KUKA KRL program: EPS_2_25990_SANMH02_A_20251014015154.src

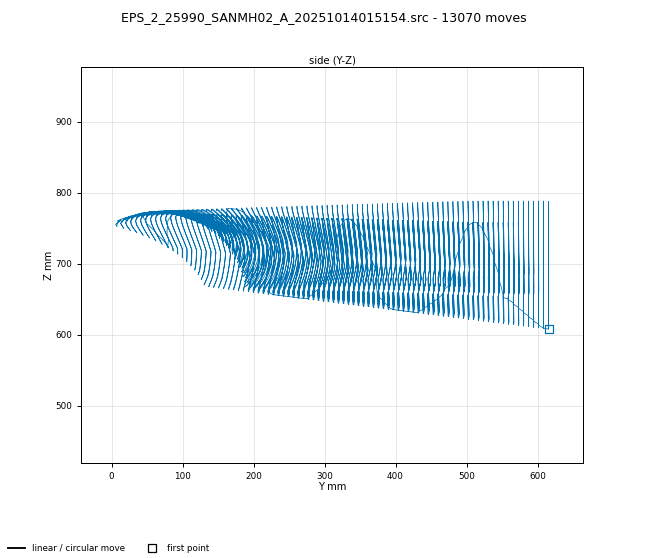
[picture p0: tool path of EPS_2_25990_SANMH02_A_20251014015154.src, 13070 of 13072 moves have a stored position in this frame; points joined in program order, loops and branches not executed]
&ACCESS RVP
&REL 4
&COMMENT QRS 19112012
&PARAM EDITMASK = *
DEF PART()
EXT BAS (BAS_COMMAND :IN,REAL :IN )
INT I
BAS (#INITMOV,0 )

;KUKA QRS Post kuka4.cps  Date:22-06-2017 !

File_ID=2883

QRS_PRE_INIT()

;Init var - Until changes are made in qrs_pre_init
Outlet_Square_prg=0
Inlet_1_Square_prg=0
Inlet_2_Square_prg=0
Inlet_3_Square_prg=0
Inlet_4_Square_prg=0
Inlet_5_Square_prg=0

Outlet_1={X 0.000, Y 504.220, Z 687.500, B 0.000, E1 0.000 }
Inlet_1={X 0.000, Y 506.400, Z 657.500, B 0.000, E1 135.000 }
Inlet_2={X 0.000, Y 506.400, Z 657.500, B 0.000, E1 224.000 }
Outlet_1_type=201
Inlet_1_type=201
Inlet_2_type=201
;QRS#1=Sidecore dimensions
;QRS#2=200-8" PVC SDR 35
;QRS#3=200-8" PVC SDR 35
;QRS#4=200-8" PVC SDR 35
;QRS#5=
;QRS#6=
;QRS#7=
;QRS#8=
;QRS#9=12-08 PSX
;QRS#10=12-08 PSX
;QRS#11=12-08 PSX
;QRS#12=
;QRS#13=
;QRS#14=
;QRS#15=
;QRS#16=1220x127x1067 3,5'
;QRS#17=EPS Height
;QRS#18=788
;QRS#19=*
;QRS#20= UPDATED VERSION 22-06-2017
;QRS#21=*
Outlet_Square=0100
Inlet_1_Square=0100
Inlet_2_Square=0100
Inlet_3_Square=0
Inlet_4_Square=0
Inlet_5_Square=0
Mill_Square=1
Outlet_Square_Prg=204
Inlet_1_Square_prg=204
Inlet_2_Square_prg=204

QRS_INIT()

$ADVANCE=5

; T1
PTP {E1 173.417,E2 173.417}
PTP {X 0,Y 615.493,A -85,B 0,C 180,E1 173.417,E2 173.417,E3 0,E4 0,E5 0,E6 0}
QRS_SPEED_INIT()
LIN {X 0,Y 615.493,Z 607.697,A -85,B 0,C 180,E1 173.417,E2 173.417,E3 0,E4 0,E5 0,E6 0} C_VEL
LIN {X 0,Y 615.492,Z 607.697,A -85,B 0,C 180,E1 170.801,E2 170.801} C_VEL
LIN {X 0,Y 615.497,Z 607.973,A -85,B 0,C 180,E1 170.138,E2 170.138} C_VEL
LIN {X 0,Y 615.488,Z 612.63,A -85,B 0,C 180,E1 167.47,E2 167.47} C_VEL
LIN {X 0,Y 615.489,Z 617.473,A -85,B 0,C 180,E1 164.774,E2 164.774} C_VEL
LIN {X 0,Y 615.454,Z 622.534,A -85,B 0,C 180,E1 162.042,E2 162.042} C_VEL
LIN {X 0,Y 615.492,Z 627.771,A -85,B 0,C 180,E1 159.269,E2 159.269} C_VEL
LIN {X 0,Y 615.481,Z 633.246,A -85,B 0,C 180,E1 156.443,E2 156.443} C_VEL
LIN {X 0,Y 615.483,Z 637.503,A -85,B 0,C 180,E1 154.284,E2 154.284} C_VEL
LIN {X 0,Y 615.478,Z 642.947,A -85,B 0,C 180,E1 151.551,E2 151.551} C_VEL
LIN {X 0,Y 615.49,Z 648.292,A -85,B 0,C 180,E1 148.914,E2 148.914} C_VEL
LIN {X 0,Y 615.498,Z 653.108,A -85,B 0,C 180,E1 146.558,E2 146.558} C_VEL
LIN {X 0,Y 615.485,Z 666.029,A -85,B 0,C 180,E1 146.282,E2 146.282} C_VEL
LIN {X 0,Y 615.461,Z 679.44,A -85,B 0,C 180,E1 145.849,E2 145.849} C_VEL
LIN {X 0,Y 615.49,Z 691.789,A -85,B 0,C 180,E1 145.299,E2 145.299} C_VEL
LIN {X 0,Y 615.49,Z 702.471,A -85,B 0,C 180,E1 144.685,E2 144.685} C_VEL
LIN {X 0,Y 615.499,Z 713.776,A -85,B 0,C 180,E1 143.871,E2 143.871} C_VEL
LIN {X 0,Y 615.497,Z 722.822,A -85,B 0,C 180,E1 143.062,E2 143.062} C_VEL
LIN {X 0,Y 615.494,Z 730.883,A -85,B 0,C 180,E1 142.181,E2 142.181} C_VEL
LIN {X 0,Y 615.492,Z 738.903,A -85,B 0,C 180,E1 141.096,E2 141.096} C_VEL
LIN {X 0,Y 615.498,Z 743.907,A -85,B 0,C 180,E1 140.25,E2 140.25} C_VEL
LIN {X 0,Y 615.497,Z 748.065,A -85,B 0,C 180,E1 139.394,E2 139.394} C_VEL
LIN {X 0,Y 615.496,Z 751.443,A -85,B 0,C 180,E1 138.527,E2 138.527} C_VEL
LIN {X 0,Y 615.496,Z 754.035,A -85,B 0,C 180,E1 137.647,E2 137.647} C_VEL
LIN {X 0,Y 615.496,Z 755.878,A -85,B 0,C 180,E1 136.756,E2 136.756} C_VEL
LIN {X 0,Y 615.495,Z 757.003,A -85,B 0,C 180,E1 135.851,E2 135.851} C_VEL
LIN {X 0,Y 615.495,Z 757.387,A -85,B 0,C 180,E1 134.932,E2 134.932} C_VEL
LIN {X 0,Y 615.494,Z 756.961,A -85,B 0,C 180,E1 133.998,E2 133.998} C_VEL
LIN {X 0,Y 615.496,Z 755.701,A -85,B 0,C 180,E1 133.048,E2 133.048} C_VEL
LIN {X 0,Y 615.495,Z 753.547,A -85,B 0,C 180,E1 132.081,E2 132.081} C_VEL
LIN {X 0,Y 615.493,Z 750.396,A -85,B 0,C 180,E1 131.095,E2 131.095} C_VEL
LIN {X 0,Y 615.497,Z 746.104,A -85,B 0,C 180,E1 130.09,E2 130.09} C_VEL
LIN {X 0,Y 615.496,Z 740.461,A -85,B 0,C 180,E1 129.063,E2 129.063} C_VEL
LIN {X 0,Y 615.495,Z 733.188,A -85,B 0,C 180,E1 128.013,E2 128.013} C_VEL
LIN {X 0,Y 615.498,Z 725.187,A -85,B 0,C 180,E1 127.089,E2 127.089} C_VEL
LIN {X 0,Y 615.499,Z 716.599,A -85,B 0,C 180,E1 126.276,E2 126.276} C_VEL
LIN {X 0,Y 615.495,Z 706.81,A -85,B 0,C 180,E1 125.515,E2 125.515} C_VEL
LIN {X 0,Y 615.485,Z 695.632,A -85,B 0,C 180,E1 124.815,E2 124.815} C_VEL
LIN {X 0,Y 615.488,Z 684.664,A -85,B 0,C 180,E1 124.276,E2 124.276} C_VEL
LIN {X 0,Y 615.483,Z 673.176,A -85,B 0,C 180,E1 123.84,E2 123.84} C_VEL
LIN {X 0,Y 615.497,Z 660.612,A -85,B 0,C 180,E1 123.498,E2 123.498} C_VEL
LIN {X 0,Y 615.485,Z 653.105,A -85,B 0,C 180,E1 123.349,E2 123.349} C_VEL
LIN {X 0,Y 615.483,Z 648.137,A -85,B 0,C 180,E1 120.92,E2 120.92} C_VEL
LIN {X 0,Y 615.491,Z 643.128,A -85,B 0,C 180,E1 118.45,E2 118.45} C_VEL
LIN {X 0,Y 615.469,Z 637.683,A -85,B 0,C 180,E1 115.717,E2 115.717} C_VEL
LIN {X 0,Y 615.473,Z 633.426,A -85,B 0,C 180,E1 113.557,E2 113.557} C_VEL
LIN {X 0,Y 615.486,Z 627.944,A -85,B 0,C 180,E1 110.731,E2 110.731} C_VEL
LIN {X 0,Y 615.477,Z 622.698,A -85,B 0,C 180,E1 107.957,E2 107.957} C_VEL
LIN {X 0,Y 615.488,Z 617.637,A -85,B 0,C 180,E1 105.226,E2 105.226} C_VEL
LIN {X 0,Y 615.485,Z 612.792,A -85,B 0,C 180,E1 102.53,E2 102.53} C_VEL
LIN {X 0,Y 615.498,Z 608.124,A -85,B 0,C 180,E1 99.862,E2 99.862} C_VEL
LIN {X 0,Y 615.485,Z 607.696,A -85,B 0,C 180,E1 99.199,E2 99.199} C_VEL
LIN {X 0,Y 615.479,Z 607.699,A -85,B 0,C 180,E1 96.557,E2 96.557} C_VEL
LIN {X 0,Y 615.49,Z 607.702,A -85,B 0,C 180,E1 93.929,E2 93.929} C_VEL
LIN {X 0,Y 615.483,Z 607.699,A -85,B 0,C 180,E1 91.309,E2 91.309} C_VEL
LIN {X 0,Y 615.481,Z 607.697,A -85,B 0,C 180,E1 88.692,E2 88.692} C_VEL
LIN {X 0,Y 615.489,Z 607.696,A -85,B 0,C 180,E1 86.072,E2 86.072} C_VEL
LIN {X 0,Y 615.489,Z 607.7,A -85,B 0,C 180,E1 83.423,E2 83.423} C_VEL
LIN {X 0,Y 615.479,Z 607.698,A -85,B 0,C 180,E1 81.464,E2 81.464} C_VEL
LIN {X 0,Y 615.495,Z 608.418,A -85,B 0,C 180,E1 80.802,E2 80.802} C_VEL
LIN {X 0,Y 615.485,Z 613.216,A -85,B 0,C 180,E1 78.14,E2 78.14} C_VEL
LIN {X 0,Y 615.48,Z 618.064,A -85,B 0,C 180,E1 75.451,E2 75.451} C_VEL
LIN {X 0,Y 615.484,Z 623.118,A -85,B 0,C 180,E1 72.73,E2 72.73} C_VEL
LIN {X 0,Y 615.491,Z 628.348,A -85,B 0,C 180,E1 69.968,E2 69.968} C_VEL
LIN {X 0,Y 615.484,Z 633.814,A -85,B 0,C 180,E1 67.156,E2 67.156} C_VEL
LIN {X 0,Y 615.471,Z 639.178,A -85,B 0,C 180,E1 64.435,E2 64.435} C_VEL
LIN {X 0,Y 615.472,Z 643.891,A -85,B 0,C 180,E1 62.085,E2 62.085} C_VEL
LIN {X 0,Y 615.479,Z 648.446,A -85,B 0,C 180,E1 59.84,E2 59.84} C_VEL
LIN {X 0,Y 615.498,Z 653.106,A -85,B 0,C 180,E1 57.559,E2 57.559} C_VEL
LIN {X 0,Y 615.493,Z 667.104,A -85,B 0,C 180,E1 57.252,E2 57.252} C_VEL
LIN {X 0,Y 615.483,Z 679.089,A -85,B 0,C 180,E1 56.862,E2 56.862} C_VEL
LIN {X 0,Y 615.466,Z 690.887,A -85,B 0,C 180,E1 56.346,E2 56.346} C_VEL
LIN {X 0,Y 615.484,Z 701.885,A -85,B 0,C 180,E1 55.724,E2 55.724} C_VEL
LIN {X 0,Y 615.498,Z 712.302,A -85,B 0,C 180,E1 54.987,E2 54.987} C_VEL
LIN {X 0,Y 615.497,Z 721.763,A -85,B 0,C 180,E1 54.165,E2 54.165} C_VEL
LIN {X 0,Y 615.498,Z 729.736,A -85,B 0,C 180,E1 53.32,E2 53.32} C_VEL
LIN {X 0,Y 615.496,Z 737.019,A -85,B 0,C 180,E1 52.374,E2 52.374} C_VEL
LIN {X 0,Y 615.492,Z 743.601,A -85,B 0,C 180,E1 51.307,E2 51.307} C_VEL
LIN {X 0,Y 615.493,Z 748.682,A -85,B 0,C 180,E1 50.251,E2 50.251} C_VEL
LIN {X 0,Y 615.495,Z 751.864,A -85,B 0,C 180,E1 49.395,E2 49.395} C_VEL
LIN {X 0,Y 615.496,Z 754.342,A -85,B 0,C 180,E1 48.528,E2 48.528} C_VEL
LIN {X 0,Y 615.499,Z 756.056,A -85,B 0,C 180,E1 47.649,E2 47.649} C_VEL
LIN {X 0,Y 615.499,Z 757.068,A -85,B 0,C 180,E1 46.757,E2 46.757} C_VEL
LIN {X 0,Y 615.497,Z 757.37,A -85,B 0,C 180,E1 45.852,E2 45.852} C_VEL
LIN {X 0,Y 615.494,Z 756.911,A -85,B 0,C 180,E1 44.933,E2 44.933} C_VEL
LIN {X 0,Y 615.493,Z 755.62,A -85,B 0,C 180,E1 43.999,E2 43.999} C_VEL
LIN {X 0,Y 615.494,Z 753.462,A -85,B 0,C 180,E1 43.049,E2 43.049} C_VEL
LIN {X 0,Y 615.497,Z 750.347,A -85,B 0,C 180,E1 42.082,E2 42.082} C_VEL
LIN {X 0,Y 615.494,Z 744.938,A -85,B 0,C 180,E1 40.851,E2 40.851} C_VEL
LIN {X 0,Y 615.498,Z 738.464,A -85,B 0,C 180,E1 39.75,E2 39.75} C_VEL
LIN {X 0,Y 615.496,Z 730.594,A -85,B 0,C 180,E1 38.694,E2 38.694} C_VEL
LIN {X 0,Y 615.498,Z 721.534,A -85,B 0,C 180,E1 37.723,E2 37.723} C_VEL
LIN {X 0,Y 615.495,Z 710.854,A -85,B 0,C 180,E1 36.809,E2 36.809} C_VEL
LIN {X 0,Y 615.481,Z 700.987,A -85,B 0,C 180,E1 36.129,E2 36.129} C_VEL
LIN {X 0,Y 615.488,Z 689.855,A -85,B 0,C 180,E1 35.516,E2 35.516} C_VEL
LIN {X 0,Y 615.489,Z 676.84,A -85,B 0,C 180,E1 34.965,E2 34.965} C_VEL
LIN {X 0,Y 615.495,Z 663.969,A -85,B 0,C 180,E1 34.574,E2 34.574} C_VEL
LIN {X 0,Y 615.483,Z 653.09,A -85,B 0,C 180,E1 34.341,E2 34.341} C_VEL
LIN {X 0,Y 615.47,Z 647.66,A -85,B 0,C 180,E1 31.687,E2 31.687} C_VEL
LIN {X 0,Y 615.486,Z 641.548,A -85,B 0,C 180,E1 28.658,E2 28.658} C_VEL
LIN {X 0,Y 615.476,Z 637.141,A -85,B 0,C 180,E1 26.445,E2 26.445} C_VEL
LIN {X 0,Y 615.456,Z 632.342,A -85,B 0,C 180,E1 24.003,E2 24.003} C_VEL
LIN {X 0,Y 615.497,Z 627.372,A -85,B 0,C 180,E1 21.432,E2 21.432} C_VEL
LIN {X 0,Y 615.492,Z 622.035,A -85,B 0,C 180,E1 18.608,E2 18.608} C_VEL
LIN {X 0,Y 615.482,Z 617.056,A -85,B 0,C 180,E1 15.905,E2 15.905} C_VEL
LIN {X 0,Y 615.494,Z 612.201,A -85,B 0,C 180,E1 13.201,E2 13.201} C_VEL
LIN {X 0,Y 615.494,Z 607.912,A -85,B 0,C 180,E1 10.894,E2 10.894} C_VEL
LIN {X 0,Y 615.49,Z 607.7,A -85,B 0,C 180,E1 9.862,E2 9.862} C_VEL
LIN {X 0,Y 615.491,Z 607.697,A -85,B 0,C 180,E1 7.216,E2 7.216} C_VEL
LIN {X 0,Y 615.498,Z 607.696,A -85,B 0,C 180,E1 4.585,E2 4.585} C_VEL
LIN {X 0,Y 615.484,Z 607.7,A -85,B 0,C 180,E1 1.963,E2 1.963} C_VEL
LIN {X 0,Y 615.487,Z 607.698,A -85,B 0,C 180,E1 -0.654,E2 -0.654} C_VEL
LIN {X 0,Y 615.495,Z 607.699,A -85,B 0,C 180,E1 -3.273,E2 -3.273} C_VEL
LIN {X 0,Y 615.478,Z 607.7,A -85,B 0,C 180,E1 -5.899,E2 -5.899} C_VEL
LIN {X 0,Y 615.491,Z 607.702,A -85,B 0,C 180,E1 -8.537,E2 -8.537} C_VEL
LIN {X 0,Y 615.497,Z 607.695,A -85,B 0,C 180,E1 -11.193,E2 -11.193} C_VEL
LIN {X 0,Y 615.482,Z 607.7,A -85,B 0,C 180,E1 -13.933,E2 -13.933} C_VEL
LIN {X 0,Y 615.485,Z 607.7,A -85,B 0,C 180,E1 -16.587,E2 -16.587} C_VEL
LIN {X 0,Y 615.496,Z 607.695,A -85,B 0,C 180,E1 -19.338,E2 -19.338} C_VEL
LIN {X 0,Y 615.483,Z 607.7,A -85,B 0,C 180,E1 -22.137,E2 -22.137} C_VEL
LIN {X 0,Y 615.493,Z 607.701,A -85,B 0,C 180,E1 -24.992,E2 -24.992} C_VEL
LIN {X 0,Y 615.491,Z 607.699,A -85,B 0,C 180,E1 -27.915,E2 -27.915} C_VEL
LIN {X 0,Y 615.499,Z 607.7,A -85,B 0,C 180,E1 -30.16,E2 -30.16} C_VEL
LIN {X 0,Y 615.482,Z 607.7,A -85,B 0,C 180,E1 -32.458,E2 -32.458} C_VEL
LIN {X 0,Y 615.476,Z 607.7,A -85,B 0,C 180,E1 -34.816,E2 -34.816} C_VEL
LIN {X 0,Y 615.486,Z 607.701,A -85,B 0,C 180,E1 -37.242,E2 -37.242} C_VEL
LIN {X 0,Y 615.482,Z 607.699,A -85,B 0,C 180,E1 -40.089,E2 -40.089} C_VEL
LIN {X 0,Y 615.484,Z 607.701,A -85,B 0,C 180,E1 -42.354,E2 -42.354} C_VEL
LIN {X 0,Y 615.478,Z 607.699,A -85,B 0,C 180,E1 -45.07,E2 -45.07} C_VEL
LIN {X 0,Y 615.479,Z 607.7,A -85,B 0,C 180,E1 -47.921,E2 -47.921} C_VEL
LIN {X 0,Y 615.476,Z 607.7,A -85,B 0,C 180,E1 -50.25,E2 -50.25} C_VEL
LIN {X 0,Y 615.486,Z 607.699,A -85,B 0,C 180,E1 -53.064,E2 -53.064} C_VEL
LIN {X 0,Y 615.482,Z 607.797,A -85,B 0,C 180,E1 -54.585,E2 -54.585} C_VEL
LIN {X 0,Y 615.484,Z 616.12,A -85,B 0,C 180,E1 -57.543,E2 -57.543} C_VEL
LIN {X 0,Y 615.449,Z 623.88,A -85,B 0,C 180,E1 -60.212,E2 -60.212} C_VEL
LIN {X 0,Y 615.438,Z 630.551,A -85,B 0,C 180,E1 -62.453,E2 -62.453} C_VEL
LIN {X 0,Y 615.47,Z 638.31,A -85,B 0,C 180,E1 -65.008,E2 -65.008} C_VEL
LIN {X 0,Y 615.494,Z 647.172,A -85,B 0,C 180,E1 -67.864,E2 -67.864} C_VEL
LIN {X 0,Y 615.477,Z 656.038,A -85,B 0,C 180,E1 -70.662,E2 -70.662} C_VEL
LIN {X 0,Y 615.479,Z 664.89,A -85,B 0,C 180,E1 -73.414,E2 -73.414} C_VEL
LIN {X 0,Y 615.486,Z 673.749,A -85,B 0,C 180,E1 -76.126,E2 -76.126} C_VEL
LIN {X 0,Y 615.489,Z 681.137,A -85,B 0,C 180,E1 -78.369,E2 -78.369} C_VEL
LIN {X 0,Y 615.489,Z 694.836,A -85,B 0,C 180,E1 -78.641,E2 -78.641} C_VEL
LIN {X 0,Y 615.461,Z 707.861,A -85,B 0,C 180,E1 -79.047,E2 -79.047} C_VEL
LIN {X 0,Y 615.469,Z 719.776,A -85,B 0,C 180,E1 -79.556,E2 -79.556} C_VEL
LIN {X 0,Y 615.489,Z 730.393,A -85,B 0,C 180,E1 -80.138,E2 -80.138} C_VEL
LIN {X 0,Y 615.498,Z 741.236,A -85,B 0,C 180,E1 -80.885,E2 -80.885} C_VEL
LIN {X 0,Y 615.497,Z 751.815,A -85,B 0,C 180,E1 -81.794,E2 -81.794} C_VEL
LIN {X 0,Y 615.498,Z 759.609,A -85,B 0,C 180,E1 -82.62,E2 -82.62} C_VEL
LIN {X 0,Y 615.497,Z 767.205,A -85,B 0,C 180,E1 -83.608,E2 -83.608} C_VEL
LIN {X 0,Y 615.498,Z 774.206,A -85,B 0,C 180,E1 -84.759,E2 -84.759} C_VEL
LIN {X 0,Y 615.494,Z 778.852,A -85,B 0,C 180,E1 -85.744,E2 -85.744} C_VEL
LIN {X 0,Y 615.494,Z 782.4,A -85,B 0,C 180,E1 -86.727,E2 -86.727} C_VEL
LIN {X 0,Y 615.497,Z 784.234,A -85,B 0,C 180,E1 -87.382,E2 -87.382} C_VEL
LIN {X 0,Y 615.498,Z 785.608,A -85,B 0,C 180,E1 -88.037,E2 -88.037} C_VEL
LIN {X 0,Y 615.496,Z 787.174,A -85,B 0,C 180,E1 -89.346,E2 -89.346} C_VEL
LIN {X 0,Y 615.494,Z 787.389,A -85,B 0,C 180,E1 -90,E2 -90} C_VEL
LIN {X 0,Y 615.495,Z 786.58,A -85,B 0,C 180,E1 -91.309,E2 -91.309} C_VEL
LIN {X 0,Y 615.498,Z 785.607,A -85,B 0,C 180,E1 -91.963,E2 -91.963} C_VEL
LIN {X 0,Y 615.497,Z 784.232,A -85,B 0,C 180,E1 -92.618,E2 -92.618} C_VEL
LIN {X 0,Y 615.496,Z 781.349,A -85,B 0,C 180,E1 -93.601,E2 -93.601} C_VEL
LIN {X 0,Y 615.498,Z 777.44,A -85,B 0,C 180,E1 -94.585,E2 -94.585} C_VEL
LIN {X 0,Y 615.499,Z 772.403,A -85,B 0,C 180,E1 -95.57,E2 -95.57} C_VEL
LIN {X 0,Y 615.497,Z 765.869,A -85,B 0,C 180,E1 -96.583,E2 -96.583} C_VEL
LIN {X 0,Y 615.497,Z 758.131,A -85,B 0,C 180,E1 -97.546,E2 -97.546} C_VEL
LIN {X 0,Y 615.498,Z 750.042,A -85,B 0,C 180,E1 -98.371,E2 -98.371} C_VEL
LIN {X 0,Y 615.499,Z 740.164,A -85,B 0,C 180,E1 -99.199,E2 -99.199} C_VEL
LIN {X 0,Y 615.489,Z 728.977,A -85,B 0,C 180,E1 -99.945,E2 -99.945} C_VEL
LIN {X 0,Y 615.464,Z 718.021,A -85,B 0,C 180,E1 -100.528,E2 -100.528} C_VEL
LIN {X 0,Y 615.464,Z 705.696,A -85,B 0,C 180,E1 -101.033,E2 -101.033} C_VEL
LIN {X 0,Y 615.49,Z 693.055,A -85,B 0,C 180,E1 -101.402,E2 -101.402} C_VEL
LIN {X 0,Y 615.489,Z 681.135,A -85,B 0,C 180,E1 -101.631,E2 -101.631} C_VEL
LIN {X 0,Y 615.492,Z 672.544,A -85,B 0,C 180,E1 -104.24,E2 -104.24} C_VEL
LIN {X 0,Y 615.484,Z 663.78,A -85,B 0,C 180,E1 -106.929,E2 -106.929} C_VEL
LIN {X 0,Y 615.468,Z 654.936,A -85,B 0,C 180,E1 -109.686,E2 -109.686} C_VEL
LIN {X 0,Y 615.492,Z 646.511,A -85,B 0,C 180,E1 -112.346,E2 -112.346} C_VEL
LIN {X 0,Y 615.471,Z 638.308,A -85,B 0,C 180,E1 -114.993,E2 -114.993} C_VEL
LIN {X 0,Y 615.436,Z 630.55,A -85,B 0,C 180,E1 -117.548,E2 -117.548} C_VEL
LIN {X 0,Y 615.499,Z 622.775,A -85,B 0,C 180,E1 -120.16,E2 -120.16} C_VEL
LIN {X 0,Y 615.438,Z 615.014,A -85,B 0,C 180,E1 -122.849,E2 -122.849} C_VEL
LIN {X 0,Y 615.48,Z 607.7,A -85,B 0,C 180,E1 -125.466,E2 -125.466} C_VEL
LIN {X 0,Y 615.489,Z 607.7,A -85,B 0,C 180,E1 -128.068,E2 -128.068} C_VEL
LIN {X 0,Y 615.491,Z 607.697,A -85,B 0,C 180,E1 -130.606,E2 -130.606} C_VEL
LIN {X 0,Y 615.498,Z 607.7,A -85,B 0,C 180,E1 -133.244,E2 -133.244} C_VEL
LIN {X 0,Y 615.482,Z 607.7,A -85,B 0,C 180,E1 -136.003,E2 -136.003} C_VEL
LIN {X 0,Y 615.486,Z 607.698,A -85,B 0,C 180,E1 -138.906,E2 -138.906} C_VEL
LIN {X 0,Y 615.485,Z 607.699,A -85,B 0,C 180,E1 -141.095,E2 -141.095} C_VEL
LIN {X 0,Y 615.481,Z 607.701,A -85,B 0,C 180,E1 -143.575,E2 -143.575} C_VEL
LIN {X 0,Y 615.495,Z 607.7,A -85,B 0,C 180,E1 -146.465,E2 -146.465} C_VEL
LIN {X 0,Y 615.486,Z 607.698,A -85,B 0,C 180,E1 -149.08,E2 -149.08} C_VEL
LIN {X 0,Y 615.489,Z 607.701,A -85,B 0,C 180,E1 -151.549,E2 -151.549} C_VEL
LIN {X 0,Y 615.497,Z 607.7,A -85,B 0,C 180,E1 -154.429,E2 -154.429} C_VEL
LIN {X 0,Y 615.486,Z 607.698,A -85,B 0,C 180,E1 -157.155,E2 -157.155} C_VEL
LIN {X 0,Y 615.494,Z 607.7,A -85,B 0,C 180,E1 -159.442,E2 -159.442} C_VEL
LIN {X 0,Y 615.476,Z 607.7,A -85,B 0,C 180,E1 -162.043,E2 -162.043} C_VEL
LIN {X 0,Y 615.497,Z 607.698,A -85,B 0,C 180,E1 -164.774,E2 -164.774} C_VEL
LIN {X 0,Y 615.487,Z 607.7,A -85,B 0,C 180,E1 -167.47,E2 -167.47} C_VEL
LIN {X 0,Y 615.476,Z 607.7,A -85,B 0,C 180,E1 -170.138,E2 -170.138} C_VEL
LIN {X 0,Y 615.496,Z 607.699,A -85,B 0,C 180,E1 -172.784,E2 -172.784} C_VEL
LIN {X 0,Y 615.486,Z 607.698,A -85,B 0,C 180,E1 -175.415,E2 -175.415} C_VEL
LIN {X 0,Y 615.481,Z 607.7,A -85,B 0,C 180,E1 -178.037,E2 -178.037} C_VEL
LIN {X 0,Y 615.494,Z 607.699,A -85,B 0,C 180,E1 -180.654,E2 -180.654} C_VEL
LIN {X 0,Y 615.488,Z 607.697,A -85,B 0,C 180,E1 -183.273,E2 -183.273} C_VEL
LIN {X 0,Y 615.495,Z 607.7,A -85,B 0,C 180,E1 -185.899,E2 -185.899} C_VEL
LIN {X 0,Y 615.493,Z 607.697,A -85,B 0,C 180,E1 -186.583,E2 -186.583} C_VEL
LIN {X 0,Y 614.816,Z 607.841,A -85,B 0,C 180,E1 -187.129,E2 -187.129} C_VEL
LIN {X 0,Y 611.98,Z 608.258,A -85,B 0,C 180,E1 -188.015,E2 -188.015} C_VEL
LIN {X 0,Y 609.589,Z 608.556,A -85,B 0,C 180,E1 -188.728,E2 -188.728} C_VEL
LIN {X 0,Y 608.555,Z 608.707,A -85,B 0,C 180,E1 -189.277,E2 -189.277} C_VEL
LIN {X 0,Y 608.466,Z 608.799,A -85,B 0,C 180,E1 -189.463,E2 -189.463} C_VEL
LIN {X 0,Y 608.466,Z 609.15,A -85,B 0,C 180,E1 -189.977,E2 -189.977} C_VEL
LIN {X 0,Y 608.453,Z 613.813,A -85,B 0,C 180,E1 -192.677,E2 -192.677} C_VEL
LIN {X 0,Y 608.439,Z 618.702,A -85,B 0,C 180,E1 -195.407,E2 -195.407} C_VEL
LIN {X 0,Y 608.429,Z 623.792,A -85,B 0,C 180,E1 -198.173,E2 -198.173} C_VEL
LIN {X 0,Y 608.437,Z 629.091,A -85,B 0,C 180,E1 -200.982,E2 -200.982} C_VEL
LIN {X 0,Y 608.433,Z 633.212,A -85,B 0,C 180,E1 -203.125,E2 -203.125} C_VEL
LIN {X 0,Y 608.44,Z 638.909,A -85,B 0,C 180,E1 -206.036,E2 -206.036} C_VEL
LIN {X 0,Y 608.442,Z 644.857,A -85,B 0,C 180,E1 -209.021,E2 -209.021} C_VEL
LIN {X 0,Y 608.42,Z 649.498,A -85,B 0,C 180,E1 -211.319,E2 -211.319} C_VEL
LIN {X 0,Y 608.444,Z 653.533,A -85,B 0,C 180,E1 -213.3,E2 -213.3} C_VEL
LIN {X 0,Y 608.512,Z 669.068,A -85,B 0,C 180,E1 -213.668,E2 -213.668} C_VEL
LIN {X 0,Y 608.48,Z 681.94,A -85,B 0,C 180,E1 -214.119,E2 -214.119} C_VEL
LIN {X 0,Y 608.506,Z 694.642,A -85,B 0,C 180,E1 -214.725,E2 -214.725} C_VEL
LIN {X 0,Y 608.496,Z 705.319,A -85,B 0,C 180,E1 -215.376,E2 -215.376} C_VEL
LIN {X 0,Y 608.493,Z 716.014,A -85,B 0,C 180,E1 -216.192,E2 -216.192} C_VEL
LIN {X 0,Y 608.469,Z 726.193,A -85,B 0,C 180,E1 -217.158,E2 -217.158} C_VEL
LIN {X 0,Y 608.453,Z 733.334,A -85,B 0,C 180,E1 -217.992,E2 -217.992} C_VEL
LIN {X 0,Y 608.437,Z 741.123,A -85,B 0,C 180,E1 -219.12,E2 -219.12} C_VEL
LIN {X 0,Y 608.454,Z 747.474,A -85,B 0,C 180,E1 -220.303,E2 -220.303} C_VEL
LIN {X 0,Y 608.427,Z 751.672,A -85,B 0,C 180,E1 -221.338,E2 -221.338} C_VEL
LIN {X 0,Y 608.438,Z 754.637,A -85,B 0,C 180,E1 -222.332,E2 -222.332} C_VEL
LIN {X 0,Y 608.433,Z 756.61,A -85,B 0,C 180,E1 -223.305,E2 -223.305} C_VEL
LIN {X 0,Y 608.418,Z 757.697,A -85,B 0,C 180,E1 -224.26,E2 -224.26} C_VEL
LIN {X 0,Y 608.416,Z 757.97,A -85,B 0,C 180,E1 -225.2,E2 -225.2} C_VEL
LIN {X 0,Y 608.428,Z 757.468,A -85,B 0,C 180,E1 -226.127,E2 -226.127} C_VEL
LIN {X 0,Y 608.436,Z 756.189,A -85,B 0,C 180,E1 -227.039,E2 -227.039} C_VEL
LIN {X 0,Y 608.425,Z 754.164,A -85,B 0,C 180,E1 -227.936,E2 -227.936} C_VEL
LIN {X 0,Y 608.43,Z 751.413,A -85,B 0,C 180,E1 -228.821,E2 -228.821} C_VEL
LIN {X 0,Y 608.444,Z 746.862,A -85,B 0,C 180,E1 -229.913,E2 -229.913} C_VEL
LIN {X 0,Y 608.439,Z 740.592,A -85,B 0,C 180,E1 -231.057,E2 -231.057} C_VEL
LIN {X 0,Y 608.453,Z 734.015,A -85,B 0,C 180,E1 -232.009,E2 -232.009} C_VEL
LIN {X 0,Y 608.461,Z 725.887,A -85,B 0,C 180,E1 -232.963,E2 -232.963} C_VEL
LIN {X 0,Y 608.486,Z 715.875,A -85,B 0,C 180,E1 -233.91,E2 -233.91} C_VEL
LIN {X 0,Y 608.489,Z 705.152,A -85,B 0,C 180,E1 -234.725,E2 -234.725} C_VEL
LIN {X 0,Y 608.495,Z 693.121,A -85,B 0,C 180,E1 -235.446,E2 -235.446} C_VEL
LIN {X 0,Y 608.527,Z 681.617,A -85,B 0,C 180,E1 -235.984,E2 -235.984} C_VEL
LIN {X 0,Y 608.522,Z 668.699,A -85,B 0,C 180,E1 -236.432,E2 -236.432} C_VEL
LIN {X 0,Y 608.557,Z 655.257,A -85,B 0,C 180,E1 -236.744,E2 -236.744} C_VEL
LIN {X 0,Y 608.43,Z 653.518,A -85,B 0,C 180,E1 -236.798,E2 -236.798} C_VEL
LIN {X 0,Y 608.424,Z 648.116,A -85,B 0,C 180,E1 -239.452,E2 -239.452} C_VEL
LIN {X 0,Y 608.424,Z 642.033,A -85,B 0,C 180,E1 -242.481,E2 -242.481} C_VEL
LIN {X 0,Y 608.427,Z 636.208,A -85,B 0,C 180,E1 -245.428,E2 -245.428} C_VEL
LIN {X 0,Y 608.438,Z 630.623,A -85,B 0,C 180,E1 -248.307,E2 -248.307} C_VEL
LIN {X 0,Y 608.458,Z 624.965,A -85,B 0,C 180,E1 -251.288,E2 -251.288} C_VEL
LIN {X 0,Y 608.443,Z 620.119,A -85,B 0,C 180,E1 -253.906,E2 -253.906} C_VEL
LIN {X 0,Y 608.463,Z 615.175,A -85,B 0,C 180,E1 -256.643,E2 -256.643} C_VEL
LIN {X 0,Y 608.473,Z 610.441,A -85,B 0,C 180,E1 -259.35,E2 -259.35} C_VEL
LIN {X 0,Y 608.467,Z 609.284,A -85,B 0,C 180,E1 -260.023,E2 -260.023} C_VEL
LIN {X 0,Y 608.443,Z 608.696,A -85,B 0,C 180,E1 -260.694,E2 -260.694} C_VEL
LIN {X 0,Y 608.462,Z 608.694,A -85,B 0,C 180,E1 -263.384,E2 -263.384} C_VEL
LIN {X 0,Y 608.458,Z 608.697,A -85,B 0,C 180,E1 -266.026,E2 -266.026} C_VEL
LIN {X 0,Y 608.468,Z 608.694,A -85,B 0,C 180,E1 -268.676,E2 -268.676} C_VEL
LIN {X 0,Y 608.466,Z 608.693,A -85,B 0,C 180,E1 -271.323,E2 -271.323} C_VEL
LIN {X 0,Y 608.457,Z 608.694,A -85,B 0,C 180,E1 -273.974,E2 -273.974} C_VEL
LIN {X 0,Y 608.482,Z 608.694,A -85,B 0,C 180,E1 -276.632,E2 -276.632} C_VEL
LIN {X 0,Y 608.434,Z 608.827,A -85,B 0,C 180,E1 -278.971,E2 -278.971} C_VEL
LIN {X 0,Y 608.45,Z 613.19,A -85,B 0,C 180,E1 -281.324,E2 -281.324} C_VEL
LIN {X 0,Y 608.473,Z 618.028,A -85,B 0,C 180,E1 -284.037,E2 -284.037} C_VEL
LIN {X 0,Y 608.443,Z 623.068,A -85,B 0,C 180,E1 -286.784,E2 -286.784} C_VEL
LIN {X 0,Y 608.458,Z 628.304,A -85,B 0,C 180,E1 -289.57,E2 -289.57} C_VEL
LIN {X 0,Y 608.43,Z 633.88,A -85,B 0,C 180,E1 -292.469,E2 -292.469} C_VEL
LIN {X 0,Y 608.424,Z 639.436,A -85,B 0,C 180,E1 -295.302,E2 -295.302} C_VEL
LIN {X 0,Y 608.419,Z 643.851,A -85,B 0,C 180,E1 -297.519,E2 -297.519} C_VEL
LIN {X 0,Y 608.417,Z 648.775,A -85,B 0,C 180,E1 -299.963,E2 -299.963} C_VEL
LIN {X 0,Y 608.435,Z 653.545,A -85,B 0,C 180,E1 -302.306,E2 -302.306} C_VEL
LIN {X 0,Y 608.544,Z 668.367,A -85,B 0,C 180,E1 -302.649,E2 -302.649} C_VEL
LIN {X 0,Y 608.529,Z 680.799,A -85,B 0,C 180,E1 -303.072,E2 -303.072} C_VEL
LIN {X 0,Y 608.469,Z 691.759,A -85,B 0,C 180,E1 -303.57,E2 -303.57} C_VEL
LIN {X 0,Y 608.491,Z 702.133,A -85,B 0,C 180,E1 -304.167,E2 -304.167} C_VEL
LIN {X 0,Y 608.49,Z 712.575,A -85,B 0,C 180,E1 -304.911,E2 -304.911} C_VEL
LIN {X 0,Y 608.459,Z 721.461,A -85,B 0,C 180,E1 -305.682,E2 -305.682} C_VEL
LIN {X 0,Y 608.455,Z 729.278,A -85,B 0,C 180,E1 -306.502,E2 -306.502} C_VEL
LIN {X 0,Y 608.444,Z 737.662,A -85,B 0,C 180,E1 -307.585,E2 -307.585} C_VEL
LIN {X 0,Y 608.43,Z 743.847,A -85,B 0,C 180,E1 -308.59,E2 -308.59} C_VEL
LIN {X 0,Y 608.426,Z 748.1,A -85,B 0,C 180,E1 -309.442,E2 -309.442} C_VEL
LIN {X 0,Y 608.431,Z 751.628,A -85,B 0,C 180,E1 -310.326,E2 -310.326} C_VEL
LIN {X 0,Y 608.422,Z 754.653,A -85,B 0,C 180,E1 -311.338,E2 -311.338} C_VEL
LIN {X 0,Y 608.439,Z 756.654,A -85,B 0,C 180,E1 -312.332,E2 -312.332} C_VEL
LIN {X 0,Y 608.435,Z 757.729,A -85,B 0,C 180,E1 -313.305,E2 -313.305} C_VEL
LIN {X 0,Y 608.419,Z 757.956,A -85,B 0,C 180,E1 -314.26,E2 -314.26} C_VEL
LIN {X 0,Y 608.416,Z 757.382,A -85,B 0,C 180,E1 -315.2,E2 -315.2} C_VEL
LIN {X 0,Y 608.427,Z 756.039,A -85,B 0,C 180,E1 -316.126,E2 -316.126} C_VEL
LIN {X 0,Y 608.435,Z 753.889,A -85,B 0,C 180,E1 -317.038,E2 -317.038} C_VEL
LIN {X 0,Y 608.429,Z 750.987,A -85,B 0,C 180,E1 -317.936,E2 -317.936} C_VEL
LIN {X 0,Y 608.44,Z 746.236,A -85,B 0,C 180,E1 -319.042,E2 -319.042} C_VEL
LIN {X 0,Y 608.44,Z 740.163,A -85,B 0,C 180,E1 -320.128,E2 -320.128} C_VEL
LIN {X 0,Y 608.467,Z 733.639,A -85,B 0,C 180,E1 -321.059,E2 -321.059} C_VEL
LIN {X 0,Y 608.454,Z 725.462,A -85,B 0,C 180,E1 -322.007,E2 -322.007} C_VEL
LIN {X 0,Y 608.467,Z 715.29,A -85,B 0,C 180,E1 -322.961,E2 -322.961} C_VEL
LIN {X 0,Y 608.499,Z 705.439,A -85,B 0,C 180,E1 -323.706,E2 -323.706} C_VEL
LIN {X 0,Y 608.499,Z 695.476,A -85,B 0,C 180,E1 -324.32,E2 -324.32} C_VEL
LIN {X 0,Y 608.516,Z 683.874,A -85,B 0,C 180,E1 -324.888,E2 -324.888} C_VEL
LIN {X 0,Y 608.524,Z 671.07,A -85,B 0,C 180,E1 -325.362,E2 -325.362} C_VEL
LIN {X 0,Y 608.549,Z 658.331,A -85,B 0,C 180,E1 -325.687,E2 -325.687} C_VEL
LIN {X 0,Y 608.415,Z 653.537,A -85,B 0,C 180,E1 -325.789,E2 -325.789} C_VEL
LIN {X 0,Y 608.416,Z 647.543,A -85,B 0,C 180,E1 -328.736,E2 -328.736} C_VEL
LIN {X 0,Y 608.424,Z 642.219,A -85,B 0,C 180,E1 -331.387,E2 -331.387} C_VEL
LIN {X 0,Y 608.403,Z 637.122,A -85,B 0,C 180,E1 -333.962,E2 -333.962} C_VEL
LIN {X 0,Y 608.429,Z 631.454,A -85,B 0,C 180,E1 -336.875,E2 -336.875} C_VEL
LIN {X 0,Y 608.43,Z 626.027,A -85,B 0,C 180,E1 -339.725,E2 -339.725} C_VEL
LIN {X 0,Y 608.453,Z 620.819,A -85,B 0,C 180,E1 -342.523,E2 -342.523} C_VEL
LIN {X 0,Y 608.444,Z 615.827,A -85,B 0,C 180,E1 -345.279,E2 -345.279} C_VEL
LIN {X 0,Y 608.469,Z 610.986,A -85,B 0,C 180,E1 -348,E2 -348} C_VEL
LIN {X 0,Y 608.457,Z 608.696,A -85,B 0,C 180,E1 -349.194,E2 -349.194} C_VEL
LIN {X 0,Y 608.479,Z 608.695,A -85,B 0,C 180,E1 -352.033,E2 -352.033} C_VEL
LIN {X 0,Y 608.465,Z 608.694,A -85,B 0,C 180,E1 -354.698,E2 -354.698} C_VEL
LIN {X 0,Y 608.486,Z 608.693,A -85,B 0,C 180,E1 -357.352,E2 -357.352} C_VEL
LIN {X 0,Y 608.47,Z 608.694,A -85,B 0,C 180,E1 -360,E2 -360} C_VEL
LIN {X 0,Y 608.481,Z 608.693,A -85,B 0,C 180,E1 -362.648,E2 -362.648} C_VEL
LIN {X 0,Y 608.472,Z 608.694,A -85,B 0,C 180,E1 -365.302,E2 -365.302} C_VEL
LIN {X 0,Y 608.471,Z 608.693,A -85,B 0,C 180,E1 -367.967,E2 -367.967} C_VEL
LIN {X 0,Y 608.468,Z 608.696,A -85,B 0,C 180,E1 -370.65,E2 -370.65} C_VEL
LIN {X 0,Y 608.47,Z 608.694,A -85,B 0,C 180,E1 -373.356,E2 -373.356} C_VEL
LIN {X 0,Y 608.456,Z 608.695,A -85,B 0,C 180,E1 -376.094,E2 -376.094} C_VEL
LIN {X 0,Y 608.454,Z 608.698,A -85,B 0,C 180,E1 -378.87,E2 -378.87} C_VEL
LIN {X 0,Y 608.473,Z 608.694,A -85,B 0,C 180,E1 -381.691,E2 -381.691} C_VEL
LIN {X 0,Y 608.452,Z 608.696,A -85,B 0,C 180,E1 -384.571,E2 -384.571} C_VEL
LIN {X 0,Y 608.487,Z 608.693,A -85,B 0,C 180,E1 -387.21,E2 -387.21} C_VEL
LIN {X 0,Y 608.472,Z 608.694,A -85,B 0,C 180,E1 -389.973,E2 -389.973} C_VEL
LIN {X 0,Y 608.457,Z 608.695,A -85,B 0,C 180,E1 -392.523,E2 -392.523} C_VEL
LIN {X 0,Y 608.445,Z 608.699,A -85,B 0,C 180,E1 -395.278,E2 -395.278} C_VEL
LIN {X 0,Y 608.468,Z 608.694,A -85,B 0,C 180,E1 -397.746,E2 -397.746} C_VEL
LIN {X 0,Y 608.449,Z 608.698,A -85,B 0,C 180,E1 -400.33,E2 -400.33} C_VEL
LIN {X 0,Y 608.471,Z 608.694,A -85,B 0,C 180,E1 -403.31,E2 -403.31} C_VEL
LIN {X 0,Y 608.463,Z 608.694,A -85,B 0,C 180,E1 -406.131,E2 -406.131} C_VEL
LIN {X 0,Y 608.455,Z 608.697,A -85,B 0,C 180,E1 -408.824,E2 -408.824} C_VEL
LIN {X 0,Y 608.467,Z 608.697,A -85,B 0,C 180,E1 -411.76,E2 -411.76} C_VEL
LIN {X 0,Y 608.462,Z 608.789,A -85,B 0,C 180,E1 -414.47,E2 -414.47} C_VEL
LIN {X 0,Y 608.427,Z 615.058,A -85,B 0,C 180,E1 -416.724,E2 -416.724} C_VEL
LIN {X 0,Y 608.439,Z 621.815,A -85,B 0,C 180,E1 -419.096,E2 -419.096} C_VEL
LIN {X 0,Y 608.463,Z 629.527,A -85,B 0,C 180,E1 -421.734,E2 -421.734} C_VEL
LIN {X 0,Y 608.44,Z 637.177,A -85,B 0,C 180,E1 -424.286,E2 -424.286} C_VEL
LIN {X 0,Y 608.445,Z 645.11,A -85,B 0,C 180,E1 -426.876,E2 -426.876} C_VEL
LIN {X 0,Y 608.463,Z 654.014,A -85,B 0,C 180,E1 -429.726,E2 -429.726} C_VEL
LIN {X 0,Y 608.452,Z 662.919,A -85,B 0,C 180,E1 -432.524,E2 -432.524} C_VEL
LIN {X 0,Y 608.438,Z 671.823,A -85,B 0,C 180,E1 -435.279,E2 -435.279} C_VEL
LIN {X 0,Y 608.444,Z 681.423,A -85,B 0,C 180,E1 -438.212,E2 -438.212} C_VEL
LIN {X 0,Y 608.551,Z 682.64,A -85,B 0,C 180,E1 -438.256,E2 -438.256} C_VEL
LIN {X 0,Y 608.539,Z 695.709,A -85,B 0,C 180,E1 -438.53,E2 -438.53} C_VEL
LIN {X 0,Y 608.501,Z 708.709,A -85,B 0,C 180,E1 -438.947,E2 -438.947} C_VEL
LIN {X 0,Y 608.491,Z 719.928,A -85,B 0,C 180,E1 -439.435,E2 -439.435} C_VEL
LIN {X 0,Y 608.482,Z 730.584,A -85,B 0,C 180,E1 -440.023,E2 -440.023} C_VEL
LIN {X 0,Y 608.483,Z 741.478,A -85,B 0,C 180,E1 -440.779,E2 -440.779} C_VEL
LIN {X 0,Y 608.475,Z 752.115,A -85,B 0,C 180,E1 -441.699,E2 -441.699} C_VEL
LIN {X 0,Y 608.471,Z 759.963,A -85,B 0,C 180,E1 -442.534,E2 -442.534} C_VEL
LIN {X 0,Y 608.461,Z 767.287,A -85,B 0,C 180,E1 -443.485,E2 -443.485} C_VEL
LIN {X 0,Y 608.45,Z 772.868,A -85,B 0,C 180,E1 -444.366,E2 -444.366} C_VEL
LIN {X 0,Y 608.432,Z 777.951,A -85,B 0,C 180,E1 -445.362,E2 -445.362} C_VEL
LIN {X 0,Y 608.449,Z 781.897,A -85,B 0,C 180,E1 -446.358,E2 -446.358} C_VEL
LIN {X 0,Y 608.425,Z 784.81,A -85,B 0,C 180,E1 -447.352,E2 -447.352} C_VEL
LIN {X 0,Y 608.443,Z 786.202,A -85,B 0,C 180,E1 -448.014,E2 -448.014} C_VEL
LIN {X 0,Y 608.438,Z 787.784,A -85,B 0,C 180,E1 -449.338,E2 -449.338} C_VEL
LIN {X 0,Y 608.434,Z 788,A -85,B 0,C 180,E1 -450,E2 -450} C_VEL
LIN {X 0,Y 608.448,Z 787.183,A -85,B 0,C 180,E1 -451.324,E2 -451.324} C_VEL
LIN {X 0,Y 608.443,Z 786.201,A -85,B 0,C 180,E1 -451.986,E2 -451.986} C_VEL
LIN {X 0,Y 608.425,Z 784.808,A -85,B 0,C 180,E1 -452.649,E2 -452.649} C_VEL
LIN {X 0,Y 608.449,Z 781.895,A -85,B 0,C 180,E1 -453.643,E2 -453.643} C_VEL
LIN {X 0,Y 608.432,Z 777.949,A -85,B 0,C 180,E1 -454.638,E2 -454.638} C_VEL
LIN {X 0,Y 608.437,Z 771.875,A -85,B 0,C 180,E1 -455.801,E2 -455.801} C_VEL
LIN {X 0,Y 608.462,Z 765.233,A -85,B 0,C 180,E1 -456.8,E2 -456.8} C_VEL
LIN {X 0,Y 608.456,Z 756.987,A -85,B 0,C 180,E1 -457.8,E2 -457.8} C_VEL
LIN {X 0,Y 608.472,Z 748.533,A -85,B 0,C 180,E1 -458.636,E2 -458.636} C_VEL
LIN {X 0,Y 608.481,Z 738.087,A -85,B 0,C 180,E1 -459.474,E2 -459.474} C_VEL
LIN {X 0,Y 608.502,Z 727.752,A -85,B 0,C 180,E1 -460.145,E2 -460.145} C_VEL
LIN {X 0,Y 608.483,Z 716.343,A -85,B 0,C 180,E1 -460.737,E2 -460.737} C_VEL
LIN {X 0,Y 608.496,Z 703.989,A -85,B 0,C 180,E1 -461.222,E2 -461.222} C_VEL
LIN {X 0,Y 608.544,Z 690.429,A -85,B 0,C 180,E1 -461.597,E2 -461.597} C_VEL
LIN {X 0,Y 608.438,Z 681.491,A -85,B 0,C 180,E1 -461.768,E2 -461.768} C_VEL
LIN {X 0,Y 608.446,Z 672.934,A -85,B 0,C 180,E1 -464.38,E2 -464.38} C_VEL
LIN {X 0,Y 608.447,Z 664.03,A -85,B 0,C 180,E1 -467.13,E2 -467.13} C_VEL
LIN {X 0,Y 608.451,Z 655.126,A -85,B 0,C 180,E1 -469.922,E2 -469.922} C_VEL
LIN {X 0,Y 608.458,Z 646.222,A -85,B 0,C 180,E1 -472.764,E2 -472.764} C_VEL
LIN {X 0,Y 608.426,Z 638.43,A -85,B 0,C 180,E1 -475.302,E2 -475.302} C_VEL
LIN {X 0,Y 608.445,Z 630.638,A -85,B 0,C 180,E1 -477.892,E2 -477.892} C_VEL
LIN {X 0,Y 608.481,Z 622.847,A -85,B 0,C 180,E1 -480.544,E2 -480.544} C_VEL
LIN {X 0,Y 608.453,Z 616.169,A -85,B 0,C 180,E1 -482.88,E2 -482.88} C_VEL
LIN {X 0,Y 608.503,Z 608.94,A -85,B 0,C 180,E1 -485.477,E2 -485.477} C_VEL
LIN {X 0,Y 608.47,Z 608.694,A -85,B 0,C 180,E1 -485.682,E2 -485.682} C_VEL
LIN {X 0,Y 608.47,Z 608.696,A -85,B 0,C 180,E1 -488.24,E2 -488.24} C_VEL
LIN {X 0,Y 608.46,Z 608.696,A -85,B 0,C 180,E1 -491.342,E2 -491.342} C_VEL
LIN {X 0,Y 608.459,Z 608.698,A -85,B 0,C 180,E1 -494.264,E2 -494.264} C_VEL
LIN {X 0,Y 608.452,Z 608.696,A -85,B 0,C 180,E1 -497.04,E2 -497.04} C_VEL
LIN {X 0,Y 608.454,Z 608.696,A -85,B 0,C 180,E1 -499.697,E2 -499.697} C_VEL
LIN {X 0,Y 608.466,Z 608.696,A -85,B 0,C 180,E1 -502.253,E2 -502.253} C_VEL
LIN {X 0,Y 608.479,Z 608.693,A -85,B 0,C 180,E1 -505.091,E2 -505.091} C_VEL
LIN {X 0,Y 608.465,Z 608.694,A -85,B 0,C 180,E1 -507.905,E2 -507.905} C_VEL
LIN {X 0,Y 608.463,Z 608.695,A -85,B 0,C 180,E1 -510.22,E2 -510.22} C_VEL
LIN {X 0,Y 608.479,Z 608.693,A -85,B 0,C 180,E1 -512.793,E2 -512.793} C_VEL
LIN {X 0,Y 608.453,Z 608.698,A -85,B 0,C 180,E1 -515.429,E2 -515.429} C_VEL
LIN {X 0,Y 608.473,Z 608.694,A -85,B 0,C 180,E1 -518.309,E2 -518.309} C_VEL
LIN {X 0,Y 608.474,Z 608.693,A -85,B 0,C 180,E1 -521.283,E2 -521.283} C_VEL
LIN {X 0,Y 608.457,Z 608.695,A -85,B 0,C 180,E1 -523.906,E2 -523.906} C_VEL
LIN {X 0,Y 608.47,Z 608.696,A -85,B 0,C 180,E1 -526.644,E2 -526.644} C_VEL
LIN {X 0,Y 608.466,Z 608.694,A -85,B 0,C 180,E1 -529.35,E2 -529.35} C_VEL
LIN {X 0,Y 608.474,Z 608.693,A -85,B 0,C 180,E1 -532.033,E2 -532.033} C_VEL
LIN {X 0,Y 608.475,Z 608.695,A -85,B 0,C 180,E1 -534.698,E2 -534.698} C_VEL
LIN {X 0,Y 608.478,Z 608.693,A -85,B 0,C 180,E1 -537.352,E2 -537.352} C_VEL
LIN {X 0,Y 608.475,Z 608.694,A -85,B 0,C 180,E1 -540,E2 -540} C_VEL
LIN {X 0,Y 608.487,Z 608.693,A -85,B 0,C 180,E1 -542.648,E2 -542.648} C_VEL
LIN {X 0,Y 608.469,Z 608.694,A -85,B 0,C 180,E1 -545.302,E2 -545.302} C_VEL
LIN {X 0,Y 608.479,Z 608.694,A -85,B 0,C 180,E1 -547.967,E2 -547.967} C_VEL
LIN {X 0,Y 608.466,Z 608.799,A -85,B 0,C 180,E1 -549.463,E2 -549.463} C_VEL
LIN {X 0,Y 607.788,Z 609.42,A -85,B 0,C 180,E1 -550.012,E2 -550.012} C_VEL
LIN {X 0,Y 604.932,Z 611.097,A -85,B 0,C 180,E1 -550.896,E2 -550.896} C_VEL
LIN {X 0,Y 602.519,Z 612.579,A -85,B 0,C 180,E1 -551.604,E2 -551.604} C_VEL
LIN {X 0,Y 601.475,Z 613.636,A -85,B 0,C 180,E1 -552.152,E2 -552.152} C_VEL
LIN {X 0,Y 601.386,Z 613.967,A -85,B 0,C 180,E1 -552.338,E2 -552.338} C_VEL
LIN {X 0,Y 601.368,Z 618.48,A -85,B 0,C 180,E1 -554.899,E2 -554.899} C_VEL
LIN {X 0,Y 601.386,Z 623.529,A -85,B 0,C 180,E1 -557.689,E2 -557.689} C_VEL
LIN {X 0,Y 601.361,Z 628.797,A -85,B 0,C 180,E1 -560.524,E2 -560.524} C_VEL
LIN {X 0,Y 601.366,Z 634.283,A -85,B 0,C 180,E1 -563.413,E2 -563.413} C_VEL
LIN {X 0,Y 601.351,Z 640.009,A -85,B 0,C 180,E1 -566.366,E2 -566.366} C_VEL
LIN {X 0,Y 601.35,Z 645.988,A -85,B 0,C 180,E1 -569.397,E2 -569.397} C_VEL
LIN {X 0,Y 601.349,Z 652.244,A -85,B 0,C 180,E1 -572.521,E2 -572.521} C_VEL
LIN {X 0,Y 601.347,Z 653.566,A -85,B 0,C 180,E1 -573.172,E2 -573.172} C_VEL
LIN {X 0,Y 601.586,Z 661.685,A -85,B 0,C 180,E1 -573.341,E2 -573.341} C_VEL
LIN {X 0,Y 601.544,Z 674.482,A -85,B 0,C 180,E1 -573.708,E2 -573.708} C_VEL
LIN {X 0,Y 601.525,Z 686.994,A -85,B 0,C 180,E1 -574.213,E2 -574.213} C_VEL
LIN {X 0,Y 601.492,Z 698.487,A -85,B 0,C 180,E1 -574.825,E2 -574.825} C_VEL
LIN {X 0,Y 601.455,Z 709.699,A -85,B 0,C 180,E1 -575.577,E2 -575.577} C_VEL
LIN {X 0,Y 601.448,Z 719.471,A -85,B 0,C 180,E1 -576.394,E2 -576.394} C_VEL
LIN {X 0,Y 601.41,Z 728.98,A -85,B 0,C 180,E1 -577.379,E2 -577.379} C_VEL
LIN {X 0,Y 601.373,Z 737.362,A -85,B 0,C 180,E1 -578.464,E2 -578.464} C_VEL
LIN {X 0,Y 601.355,Z 743.847,A -85,B 0,C 180,E1 -579.526,E2 -579.526} C_VEL
LIN {X 0,Y 601.335,Z 748.847,A -85,B 0,C 180,E1 -580.564,E2 -580.564} C_VEL
LIN {X 0,Y 601.346,Z 753.199,A -85,B 0,C 180,E1 -581.772,E2 -581.772} C_VEL
LIN {X 0,Y 601.343,Z 755.489,A -85,B 0,C 180,E1 -582.677,E2 -582.677} C_VEL
LIN {X 0,Y 601.345,Z 757.054,A -85,B 0,C 180,E1 -583.594,E2 -583.594} C_VEL
LIN {X 0,Y 601.337,Z 757.881,A -85,B 0,C 180,E1 -584.527,E2 -584.527} C_VEL
LIN {X 0,Y 601.337,Z 757.907,A -85,B 0,C 180,E1 -585.474,E2 -585.474} C_VEL
LIN {X 0,Y 601.346,Z 757.124,A -85,B 0,C 180,E1 -586.436,E2 -586.436} C_VEL
LIN {X 0,Y 601.343,Z 755.481,A -85,B 0,C 180,E1 -587.417,E2 -587.417} C_VEL
LIN {X 0,Y 601.345,Z 752.891,A -85,B 0,C 180,E1 -588.416,E2 -588.416} C_VEL
LIN {X 0,Y 601.333,Z 749.226,A -85,B 0,C 180,E1 -589.436,E2 -589.436} C_VEL
LIN {X 0,Y 601.385,Z 743.252,A -85,B 0,C 180,E1 -590.674,E2 -590.674} C_VEL
LIN {X 0,Y 601.39,Z 736.661,A -85,B 0,C 180,E1 -591.73,E2 -591.73} C_VEL
LIN {X 0,Y 601.402,Z 728.105,A -85,B 0,C 180,E1 -592.811,E2 -592.811} C_VEL
LIN {X 0,Y 601.442,Z 719.061,A -85,B 0,C 180,E1 -593.735,E2 -593.735} C_VEL
LIN {X 0,Y 601.464,Z 708.563,A -85,B 0,C 180,E1 -594.595,E2 -594.595} C_VEL
LIN {X 0,Y 601.483,Z 698.302,A -85,B 0,C 180,E1 -595.276,E2 -595.276} C_VEL
LIN {X 0,Y 601.522,Z 686.767,A -85,B 0,C 180,E1 -595.888,E2 -595.888} C_VEL
LIN {X 0,Y 601.567,Z 674.105,A -85,B 0,C 180,E1 -596.394,E2 -596.394} C_VEL
LIN {X 0,Y 601.59,Z 661.218,A -85,B 0,C 180,E1 -596.76,E2 -596.76} C_VEL
LIN {X 0,Y 601.356,Z 653.841,A -85,B 0,C 180,E1 -596.913,E2 -596.913} C_VEL
LIN {X 0,Y 601.343,Z 653.529,A -85,B 0,C 180,E1 -596.933,E2 -596.933} C_VEL
LIN {X 0,Y 601.349,Z 647.638,A -85,B 0,C 180,E1 -599.865,E2 -599.865} C_VEL
LIN {X 0,Y 601.34,Z 641.658,A -85,B 0,C 180,E1 -602.883,E2 -602.883} C_VEL
LIN {X 0,Y 601.363,Z 636.12,A -85,B 0,C 180,E1 -605.724,E2 -605.724} C_VEL
LIN {X 0,Y 601.351,Z 631.684,A -85,B 0,C 180,E1 -608.038,E2 -608.038} C_VEL
LIN {X 0,Y 601.375,Z 626.303,A -85,B 0,C 180,E1 -610.899,E2 -610.899} C_VEL
LIN {X 0,Y 601.393,Z 621.723,A -85,B 0,C 180,E1 -613.39,E2 -613.39} C_VEL
LIN {X 0,Y 601.41,Z 616.183,A -85,B 0,C 180,E1 -616.484,E2 -616.484} C_VEL
LIN {X 0,Y 601.421,Z 611.463,A -85,B 0,C 180,E1 -619.224,E2 -619.224} C_VEL
LIN {X 0,Y 601.409,Z 610.296,A -85,B 0,C 180,E1 -619.904,E2 -619.904} C_VEL
LIN {X 0,Y 601.385,Z 609.575,A -85,B 0,C 180,E1 -620.583,E2 -620.583} C_VEL
LIN {X 0,Y 601.448,Z 609.57,A -85,B 0,C 180,E1 -622.615,E2 -622.615} C_VEL
LIN {X 0,Y 601.417,Z 609.571,A -85,B 0,C 180,E1 -625.308,E2 -625.308} C_VEL
LIN {X 0,Y 601.436,Z 609.568,A -85,B 0,C 180,E1 -627.991,E2 -627.991} C_VEL
LIN {X 0,Y 601.456,Z 609.568,A -85,B 0,C 180,E1 -630.669,E2 -630.669} C_VEL
LIN {X 0,Y 601.435,Z 609.57,A -85,B 0,C 180,E1 -633.349,E2 -633.349} C_VEL
LIN {X 0,Y 601.42,Z 609.57,A -85,B 0,C 180,E1 -636.037,E2 -636.037} C_VEL
LIN {X 0,Y 601.403,Z 609.574,A -85,B 0,C 180,E1 -638.738,E2 -638.738} C_VEL
LIN {X 0,Y 601.367,Z 609.636,A -85,B 0,C 180,E1 -639.077,E2 -639.077} C_VEL
LIN {X 0,Y 601.386,Z 614.176,A -85,B 0,C 180,E1 -641.459,E2 -641.459} C_VEL
LIN {X 0,Y 601.402,Z 619.025,A -85,B 0,C 180,E1 -644.205,E2 -644.205} C_VEL
LIN {X 0,Y 601.365,Z 624.08,A -85,B 0,C 180,E1 -646.987,E2 -646.987} C_VEL
LIN {X 0,Y 601.377,Z 629.333,A -85,B 0,C 180,E1 -649.81,E2 -649.81} C_VEL
LIN {X 0,Y 601.366,Z 634.805,A -85,B 0,C 180,E1 -652.684,E2 -652.684} C_VEL
LIN {X 0,Y 601.345,Z 639.061,A -85,B 0,C 180,E1 -654.881,E2 -654.881} C_VEL
LIN {X 0,Y 601.346,Z 643.91,A -85,B 0,C 180,E1 -657.349,E2 -657.349} C_VEL
LIN {X 0,Y 601.339,Z 649.526,A -85,B 0,C 180,E1 -660.168,E2 -660.168} C_VEL
LIN {X 0,Y 601.343,Z 653.577,A -85,B 0,C 180,E1 -662.174,E2 -662.174} C_VEL
LIN {X 0,Y 601.595,Z 661.796,A -85,B 0,C 180,E1 -662.344,E2 -662.344} C_VEL
LIN {X 0,Y 601.557,Z 674.056,A -85,B 0,C 180,E1 -662.694,E2 -662.694} C_VEL
LIN {X 0,Y 601.52,Z 686.152,A -85,B 0,C 180,E1 -663.174,E2 -663.174} C_VEL
LIN {X 0,Y 601.456,Z 697.976,A -85,B 0,C 180,E1 -663.793,E2 -663.793} C_VEL
LIN {X 0,Y 601.441,Z 708.95,A -85,B 0,C 180,E1 -664.522,E2 -664.522} C_VEL
LIN {X 0,Y 601.425,Z 718.551,A -85,B 0,C 180,E1 -665.309,E2 -665.309} C_VEL
LIN {X 0,Y 601.387,Z 727.919,A -85,B 0,C 180,E1 -666.258,E2 -666.258} C_VEL
LIN {X 0,Y 601.383,Z 735.308,A -85,B 0,C 180,E1 -667.175,E2 -667.175} C_VEL
LIN {X 0,Y 601.356,Z 742.458,A -85,B 0,C 180,E1 -668.272,E2 -668.272} C_VEL
LIN {X 0,Y 601.333,Z 746.923,A -85,B 0,C 180,E1 -669.132,E2 -669.132} C_VEL
LIN {X 0,Y 601.354,Z 750.586,A -85,B 0,C 180,E1 -669.999,E2 -669.999} C_VEL
LIN {X 0,Y 601.329,Z 753.529,A -85,B 0,C 180,E1 -670.881,E2 -670.881} C_VEL
LIN {X 0,Y 601.324,Z 755.693,A -85,B 0,C 180,E1 -671.773,E2 -671.773} C_VEL
LIN {X 0,Y 601.342,Z 757.148,A -85,B 0,C 180,E1 -672.676,E2 -672.676} C_VEL
LIN {X 0,Y 601.343,Z 757.901,A -85,B 0,C 180,E1 -673.593,E2 -673.593} C_VEL
LIN {X 0,Y 601.333,Z 757.89,A -85,B 0,C 180,E1 -674.526,E2 -674.526} C_VEL
LIN {X 0,Y 601.333,Z 757.08,A -85,B 0,C 180,E1 -675.473,E2 -675.473} C_VEL
LIN {X 0,Y 601.342,Z 755.44,A -85,B 0,C 180,E1 -676.435,E2 -676.435} C_VEL
LIN {X 0,Y 601.341,Z 752.886,A -85,B 0,C 180,E1 -677.416,E2 -677.416} C_VEL
LIN {X 0,Y 601.348,Z 749.313,A -85,B 0,C 180,E1 -678.414,E2 -678.414} C_VEL
LIN {X 0,Y 601.348,Z 744.55,A -85,B 0,C 180,E1 -679.433,E2 -679.433} C_VEL
LIN {X 0,Y 601.372,Z 738.391,A -85,B 0,C 180,E1 -680.471,E2 -680.471} C_VEL
LIN {X 0,Y 601.377,Z 730.495,A -85,B 0,C 180,E1 -681.535,E2 -681.535} C_VEL
LIN {X 0,Y 601.432,Z 721.785,A -85,B 0,C 180,E1 -682.475,E2 -682.475} C_VEL
LIN {X 0,Y 601.468,Z 712.197,A -85,B 0,C 180,E1 -683.317,E2 -683.317} C_VEL
LIN {X 0,Y 601.448,Z 701.687,A -85,B 0,C 180,E1 -684.069,E2 -684.069} C_VEL
LIN {X 0,Y 601.524,Z 690.826,A -85,B 0,C 180,E1 -684.69,E2 -684.69} C_VEL
LIN {X 0,Y 601.544,Z 678.655,A -85,B 0,C 180,E1 -685.229,E2 -685.229} C_VEL
LIN {X 0,Y 601.582,Z 665.659,A -85,B 0,C 180,E1 -685.651,E2 -685.651} C_VEL
LIN {X 0,Y 601.435,Z 654.552,A -85,B 0,C 180,E1 -685.898,E2 -685.898} C_VEL
LIN {X 0,Y 601.349,Z 653.515,A -85,B 0,C 180,E1 -685.94,E2 -685.94} C_VEL
LIN {X 0,Y 601.321,Z 648.249,A -85,B 0,C 180,E1 -688.56,E2 -688.56} C_VEL
LIN {X 0,Y 601.337,Z 642.672,A -85,B 0,C 180,E1 -691.368,E2 -691.368} C_VEL
LIN {X 0,Y 601.344,Z 637.241,A -85,B 0,C 180,E1 -694.145,E2 -694.145} C_VEL
LIN {X 0,Y 601.356,Z 632.543,A -85,B 0,C 180,E1 -696.587,E2 -696.587} C_VEL
LIN {X 0,Y 601.363,Z 627.093,A -85,B 0,C 180,E1 -699.476,E2 -699.476} C_VEL
LIN {X 0,Y 601.394,Z 621.866,A -85,B 0,C 180,E1 -702.311,E2 -702.311} C_VEL
LIN {X 0,Y 601.373,Z 616.862,A -85,B 0,C 180,E1 -705.102,E2 -705.102} C_VEL
LIN {X 0,Y 601.382,Z 613.149,A -85,B 0,C 180,E1 -707.171,E2 -707.171} C_VEL
LIN {X 0,Y 601.385,Z 609.579,A -85,B 0,C 180,E1 -709.005,E2 -709.005} C_VEL
LIN {X 0,Y 601.439,Z 609.57,A -85,B 0,C 180,E1 -711.262,E2 -711.262} C_VEL
LIN {X 0,Y 601.421,Z 609.573,A -85,B 0,C 180,E1 -713.963,E2 -713.963} C_VEL
LIN {X 0,Y 601.432,Z 609.57,A -85,B 0,C 180,E1 -716.65,E2 -716.65} C_VEL
LIN {X 0,Y 601.458,Z 609.569,A -85,B 0,C 180,E1 -719.33,E2 -719.33} C_VEL
LIN {X 0,Y 601.417,Z 609.572,A -85,B 0,C 180,E1 -722.009,E2 -722.009} C_VEL
LIN {X 0,Y 601.429,Z 609.571,A -85,B 0,C 180,E1 -724.692,E2 -724.692} C_VEL
LIN {X 0,Y 601.454,Z 609.569,A -85,B 0,C 180,E1 -727.385,E2 -727.385} C_VEL
LIN {X 0,Y 601.429,Z 609.57,A -85,B 0,C 180,E1 -730.095,E2 -730.095} C_VEL
LIN {X 0,Y 601.425,Z 609.572,A -85,B 0,C 180,E1 -732.828,E2 -732.828} C_VEL
LIN {X 0,Y 601.418,Z 609.573,A -85,B 0,C 180,E1 -735.591,E2 -735.591} C_VEL
LIN {X 0,Y 601.418,Z 609.572,A -85,B 0,C 180,E1 -738.392,E2 -738.392} C_VEL
LIN {X 0,Y 601.41,Z 609.573,A -85,B 0,C 180,E1 -741.239,E2 -741.239} C_VEL
LIN {X 0,Y 601.457,Z 609.568,A -85,B 0,C 180,E1 -744.14,E2 -744.14} C_VEL
LIN {X 0,Y 601.457,Z 609.569,A -85,B 0,C 180,E1 -747.111,E2 -747.111} C_VEL
LIN {X 0,Y 601.446,Z 609.571,A -85,B 0,C 180,E1 -750.163,E2 -750.163} C_VEL
LIN {X 0,Y 601.42,Z 609.571,A -85,B 0,C 180,E1 -752.716,E2 -752.716} C_VEL
LIN {X 0,Y 601.396,Z 609.576,A -85,B 0,C 180,E1 -755.113,E2 -755.113} C_VEL
LIN {X 0,Y 601.432,Z 609.572,A -85,B 0,C 180,E1 -757.419,E2 -757.419} C_VEL
LIN {X 0,Y 601.409,Z 609.573,A -85,B 0,C 180,E1 -759.995,E2 -759.995} C_VEL
LIN {X 0,Y 601.407,Z 609.574,A -85,B 0,C 180,E1 -762.671,E2 -762.671} C_VEL
LIN {X 0,Y 601.424,Z 609.573,A -85,B 0,C 180,E1 -765.483,E2 -765.483} C_VEL
LIN {X 0,Y 601.423,Z 609.572,A -85,B 0,C 180,E1 -768.407,E2 -768.407} C_VEL
LIN {X 0,Y 601.433,Z 609.571,A -85,B 0,C 180,E1 -771.529,E2 -771.529} C_VEL
LIN {X 0,Y 601.452,Z 609.717,A -85,B 0,C 180,E1 -774.336,E2 -774.336} C_VEL
LIN {X 0,Y 601.493,Z 614.413,A -85,B 0,C 180,E1 -776.056,E2 -776.056} C_VEL
LIN {X 0,Y 601.427,Z 621.386,A -85,B 0,C 180,E1 -778.545,E2 -778.545} C_VEL
LIN {X 0,Y 601.465,Z 629.527,A -85,B 0,C 180,E1 -781.375,E2 -781.375} C_VEL
LIN {X 0,Y 601.406,Z 637.691,A -85,B 0,C 180,E1 -784.134,E2 -784.134} C_VEL
LIN {X 0,Y 601.396,Z 645.11,A -85,B 0,C 180,E1 -786.589,E2 -786.589} C_VEL
LIN {X 0,Y 601.412,Z 654.014,A -85,B 0,C 180,E1 -789.478,E2 -789.478} C_VEL
LIN {X 0,Y 601.394,Z 662.919,A -85,B 0,C 180,E1 -792.312,E2 -792.312} C_VEL
LIN {X 0,Y 601.363,Z 671.823,A -85,B 0,C 180,E1 -795.102,E2 -795.102} C_VEL
LIN {X 0,Y 601.363,Z 680.728,A -85,B 0,C 180,E1 -797.857,E2 -797.857} C_VEL
LIN {X 0,Y 601.383,Z 681.493,A -85,B 0,C 180,E1 -798.093,E2 -798.093} C_VEL
LIN {X 0,Y 601.594,Z 694.946,A -85,B 0,C 180,E1 -798.375,E2 -798.375} C_VEL
LIN {X 0,Y 601.548,Z 707.21,A -85,B 0,C 180,E1 -798.761,E2 -798.761} C_VEL
LIN {X 0,Y 601.495,Z 719.93,A -85,B 0,C 180,E1 -799.311,E2 -799.311} C_VEL
LIN {X 0,Y 601.486,Z 730.585,A -85,B 0,C 180,E1 -799.906,E2 -799.906} C_VEL
LIN {X 0,Y 601.449,Z 741.479,A -85,B 0,C 180,E1 -800.67,E2 -800.67} C_VEL
LIN {X 0,Y 601.429,Z 752.115,A -85,B 0,C 180,E1 -801.601,E2 -801.601} C_VEL
LIN {X 0,Y 601.418,Z 759.963,A -85,B 0,C 180,E1 -802.446,E2 -802.446} C_VEL
LIN {X 0,Y 601.37,Z 767.225,A -85,B 0,C 180,E1 -803.398,E2 -803.398} C_VEL
LIN {X 0,Y 601.371,Z 772.868,A -85,B 0,C 180,E1 -804.299,E2 -804.299} C_VEL
LIN {X 0,Y 601.336,Z 777.951,A -85,B 0,C 180,E1 -805.308,E2 -805.308} C_VEL
LIN {X 0,Y 601.368,Z 781.897,A -85,B 0,C 180,E1 -806.315,E2 -806.315} C_VEL
LIN {X 0,Y 601.325,Z 784.81,A -85,B 0,C 180,E1 -807.321,E2 -807.321} C_VEL
LIN {X 0,Y 601.342,Z 786.202,A -85,B 0,C 180,E1 -807.991,E2 -807.991} C_VEL
LIN {X 0,Y 601.339,Z 787.784,A -85,B 0,C 180,E1 -809.331,E2 -809.331} C_VEL
LIN {X 0,Y 601.335,Z 788,A -85,B 0,C 180,E1 -810,E2 -810} C_VEL
LIN {X 0,Y 601.347,Z 787.184,A -85,B 0,C 180,E1 -811.34,E2 -811.34} C_VEL
LIN {X 0,Y 601.342,Z 786.201,A -85,B 0,C 180,E1 -812.01,E2 -812.01} C_VEL
LIN {X 0,Y 601.325,Z 784.809,A -85,B 0,C 180,E1 -812.68,E2 -812.68} C_VEL
LIN {X 0,Y 601.368,Z 781.895,A -85,B 0,C 180,E1 -813.686,E2 -813.686} C_VEL
LIN {X 0,Y 601.336,Z 777.949,A -85,B 0,C 180,E1 -814.693,E2 -814.693} C_VEL
LIN {X 0,Y 601.372,Z 771.875,A -85,B 0,C 180,E1 -815.869,E2 -815.869} C_VEL
LIN {X 0,Y 601.382,Z 765.233,A -85,B 0,C 180,E1 -816.88,E2 -816.88} C_VEL
LIN {X 0,Y 601.401,Z 756.987,A -85,B 0,C 180,E1 -817.893,E2 -817.893} C_VEL
LIN {X 0,Y 601.436,Z 748.534,A -85,B 0,C 180,E1 -818.738,E2 -818.738} C_VEL
LIN {X 0,Y 601.451,Z 738.088,A -85,B 0,C 180,E1 -819.585,E2 -819.585} C_VEL
LIN {X 0,Y 601.486,Z 727.753,A -85,B 0,C 180,E1 -820.264,E2 -820.264} C_VEL
LIN {X 0,Y 601.494,Z 716.096,A -85,B 0,C 180,E1 -820.875,E2 -820.875} C_VEL
LIN {X 0,Y 601.524,Z 703.304,A -85,B 0,C 180,E1 -821.376,E2 -821.376} C_VEL
LIN {X 0,Y 601.587,Z 690.428,A -85,B 0,C 180,E1 -821.733,E2 -821.733} C_VEL
LIN {X 0,Y 601.383,Z 681.491,A -85,B 0,C 180,E1 -821.908,E2 -821.908} C_VEL
LIN {X 0,Y 601.388,Z 672.934,A -85,B 0,C 180,E1 -824.552,E2 -824.552} C_VEL
LIN {X 0,Y 601.388,Z 664.03,A -85,B 0,C 180,E1 -827.338,E2 -827.338} C_VEL
LIN {X 0,Y 601.397,Z 655.126,A -85,B 0,C 180,E1 -830.166,E2 -830.166} C_VEL
LIN {X 0,Y 601.419,Z 646.221,A -85,B 0,C 180,E1 -833.046,E2 -833.046} C_VEL
LIN {X 0,Y 601.407,Z 638.43,A -85,B 0,C 180,E1 -835.619,E2 -835.619} C_VEL
LIN {X 0,Y 601.451,Z 630.638,A -85,B 0,C 180,E1 -838.245,E2 -838.245} C_VEL
LIN {X 0,Y 601.43,Z 622.847,A -85,B 0,C 180,E1 -840.942,E2 -840.942} C_VEL
LIN {X 0,Y 601.45,Z 616.157,A -85,B 0,C 180,E1 -843.312,E2 -843.312} C_VEL
LIN {X 0,Y 601.47,Z 609.953,A -85,B 0,C 180,E1 -845.577,E2 -845.577} C_VEL
LIN {X 0,Y 601.419,Z 609.573,A -85,B 0,C 180,E1 -845.753,E2 -845.753} C_VEL
LIN {X 0,Y 601.437,Z 609.57,A -85,B 0,C 180,E1 -848.471,E2 -848.471} C_VEL
LIN {X 0,Y 601.425,Z 609.571,A -85,B 0,C 180,E1 -851.593,E2 -851.593} C_VEL
LIN {X 0,Y 601.429,Z 609.571,A -85,B 0,C 180,E1 -854.518,E2 -854.518} C_VEL
LIN {X 0,Y 601.41,Z 609.575,A -85,B 0,C 180,E1 -857.41,E2 -857.41} C_VEL
LIN {X 0,Y 601.444,Z 609.57,A -85,B 0,C 180,E1 -860.464,E2 -860.464} C_VEL
LIN {X 0,Y 601.404,Z 609.576,A -85,B 0,C 180,E1 -863.417,E2 -863.417} C_VEL
LIN {X 0,Y 601.436,Z 609.57,A -85,B 0,C 180,E1 -866.064,E2 -866.064} C_VEL
LIN {X 0,Y 601.443,Z 609.57,A -85,B 0,C 180,E1 -868.542,E2 -868.542} C_VEL
LIN {X 0,Y 601.434,Z 609.572,A -85,B 0,C 180,E1 -871.373,E2 -871.373} C_VEL
LIN {X 0,Y 601.403,Z 609.575,A -85,B 0,C 180,E1 -873.636,E2 -873.636} C_VEL
LIN {X 0,Y 601.42,Z 609.574,A -85,B 0,C 180,E1 -876.59,E2 -876.59} C_VEL
LIN {X 0,Y 601.434,Z 609.572,A -85,B 0,C 180,E1 -879.478,E2 -879.478} C_VEL
LIN {X 0,Y 601.399,Z 609.575,A -85,B 0,C 180,E1 -882.312,E2 -882.312} C_VEL
LIN {X 0,Y 601.417,Z 609.573,A -85,B 0,C 180,E1 -884.409,E2 -884.409} C_VEL
LIN {X 0,Y 601.425,Z 609.571,A -85,B 0,C 180,E1 -887.172,E2 -887.172} C_VEL
LIN {X 0,Y 601.429,Z 609.571,A -85,B 0,C 180,E1 -889.905,E2 -889.905} C_VEL
LIN {X 0,Y 601.457,Z 609.569,A -85,B 0,C 180,E1 -892.615,E2 -892.615} C_VEL
LIN {X 0,Y 601.425,Z 609.571,A -85,B 0,C 180,E1 -895.308,E2 -895.308} C_VEL
LIN {X 0,Y 601.422,Z 609.572,A -85,B 0,C 180,E1 -897.991,E2 -897.991} C_VEL
LIN {X 0,Y 601.458,Z 609.568,A -85,B 0,C 180,E1 -900.67,E2 -900.67} C_VEL
LIN {X 0,Y 601.432,Z 609.57,A -85,B 0,C 180,E1 -903.35,E2 -903.35} C_VEL
LIN {X 0,Y 601.421,Z 609.573,A -85,B 0,C 180,E1 -906.037,E2 -906.037} C_VEL
LIN {X 0,Y 601.44,Z 609.571,A -85,B 0,C 180,E1 -908.738,E2 -908.738} C_VEL
LIN {X 0,Y 601.413,Z 609.606,A -85,B 0,C 180,E1 -909.453,E2 -909.453} C_VEL
LIN {X 0,Y 601.421,Z 610.196,A -85,B 0,C 180,E1 -910.095,E2 -910.095} C_VEL
LIN {X 0,Y 601.386,Z 613.967,A -85,B 0,C 180,E1 -912.338,E2 -912.338} C_VEL
LIN {X 0,Y 600.709,Z 614.997,A -85,B 0,C 180,E1 -912.888,E2 -912.888} C_VEL
LIN {X 0,Y 597.852,Z 616.851,A -85,B 0,C 180,E1 -913.779,E2 -913.779} C_VEL
LIN {X 0,Y 595.434,Z 618.354,A -85,B 0,C 180,E1 -914.495,E2 -914.495} C_VEL
LIN {X 0,Y 594.383,Z 619.435,A -85,B 0,C 180,E1 -915.048,E2 -915.048} C_VEL
LIN {X 0,Y 594.291,Z 619.776,A -85,B 0,C 180,E1 -915.236,E2 -915.236} C_VEL
LIN {X 0,Y 594.305,Z 624.565,A -85,B 0,C 180,E1 -917.907,E2 -917.907} C_VEL
LIN {X 0,Y 594.312,Z 630.07,A -85,B 0,C 180,E1 -920.899,E2 -920.899} C_VEL
LIN {X 0,Y 594.267,Z 635.361,A -85,B 0,C 180,E1 -923.709,E2 -923.709} C_VEL
LIN {X 0,Y 594.264,Z 641.112,A -85,B 0,C 180,E1 -926.706,E2 -926.706} C_VEL
LIN {X 0,Y 594.257,Z 645.596,A -85,B 0,C 180,E1 -929.005,E2 -929.005} C_VEL
LIN {X 0,Y 594.228,Z 650.755,A -85,B 0,C 180,E1 -931.619,E2 -931.619} C_VEL
LIN {X 0,Y 594.278,Z 653.541,A -85,B 0,C 180,E1 -933.02,E2 -933.02} C_VEL
LIN {X 0,Y 594.677,Z 658.661,A -85,B 0,C 180,E1 -933.134,E2 -933.134} C_VEL
LIN {X 0,Y 594.6,Z 670.542,A -85,B 0,C 180,E1 -933.442,E2 -933.442} C_VEL
LIN {X 0,Y 594.543,Z 682.751,A -85,B 0,C 180,E1 -933.895,E2 -933.895} C_VEL
LIN {X 0,Y 594.485,Z 695.146,A -85,B 0,C 180,E1 -934.507,E2 -934.507} C_VEL
LIN {X 0,Y 594.468,Z 705.567,A -85,B 0,C 180,E1 -935.162,E2 -935.162} C_VEL
LIN {X 0,Y 594.418,Z 715.396,A -85,B 0,C 180,E1 -935.926,E2 -935.926} C_VEL
LIN {X 0,Y 594.332,Z 724.211,A -85,B 0,C 180,E1 -936.761,E2 -936.761} C_VEL
LIN {X 0,Y 594.298,Z 732.743,A -85,B 0,C 180,E1 -937.748,E2 -937.748} C_VEL
LIN {X 0,Y 594.301,Z 740.133,A -85,B 0,C 180,E1 -938.812,E2 -938.812} C_VEL
LIN {X 0,Y 594.283,Z 745.448,A -85,B 0,C 180,E1 -939.764,E2 -939.764} C_VEL
LIN {X 0,Y 594.237,Z 750.059,A -85,B 0,C 180,E1 -940.806,E2 -940.806} C_VEL
LIN {X 0,Y 594.269,Z 753.509,A -85,B 0,C 180,E1 -941.836,E2 -941.836} C_VEL
LIN {X 0,Y 594.249,Z 755.894,A -85,B 0,C 180,E1 -942.84,E2 -942.84} C_VEL
LIN {X 0,Y 594.233,Z 757.704,A -85,B 0,C 180,E1 -944.251,E2 -944.251} C_VEL
LIN {X 0,Y 594.223,Z 757.969,A -85,B 0,C 180,E1 -945.205,E2 -945.205} C_VEL
LIN {X 0,Y 594.238,Z 757.445,A -85,B 0,C 180,E1 -946.174,E2 -946.174} C_VEL
LIN {X 0,Y 594.249,Z 756.065,A -85,B 0,C 180,E1 -947.16,E2 -947.16} C_VEL
LIN {X 0,Y 594.241,Z 752.679,A -85,B 0,C 180,E1 -948.524,E2 -948.524} C_VEL
LIN {X 0,Y 594.254,Z 749.498,A -85,B 0,C 180,E1 -949.423,E2 -949.423} C_VEL
LIN {X 0,Y 594.294,Z 744.366,A -85,B 0,C 180,E1 -950.533,E2 -950.533} C_VEL
LIN {X 0,Y 594.298,Z 737.532,A -85,B 0,C 180,E1 -951.679,E2 -951.679} C_VEL
LIN {X 0,Y 594.33,Z 730.225,A -85,B 0,C 180,E1 -952.658,E2 -952.658} C_VEL
LIN {X 0,Y 594.388,Z 721.117,A -85,B 0,C 180,E1 -953.64,E2 -953.64} C_VEL
LIN {X 0,Y 594.421,Z 711.416,A -85,B 0,C 180,E1 -954.492,E2 -954.492} C_VEL
LIN {X 0,Y 594.462,Z 701.225,A -85,B 0,C 180,E1 -955.219,E2 -955.219} C_VEL
LIN {X 0,Y 594.543,Z 690.37,A -85,B 0,C 180,E1 -955.839,E2 -955.839} C_VEL
LIN {X 0,Y 594.573,Z 677.57,A -85,B 0,C 180,E1 -956.404,E2 -956.404} C_VEL
LIN {X 0,Y 594.657,Z 664.701,A -85,B 0,C 180,E1 -956.815,E2 -956.815} C_VEL
LIN {X 0,Y 594.45,Z 655.081,A -85,B 0,C 180,E1 -957.029,E2 -957.029} C_VEL
LIN {X 0,Y 594.258,Z 653.532,A -85,B 0,C 180,E1 -957.075,E2 -957.075} C_VEL
LIN {X 0,Y 594.243,Z 648.329,A -85,B 0,C 180,E1 -959.696,E2 -959.696} C_VEL
LIN {X 0,Y 594.265,Z 642.765,A -85,B 0,C 180,E1 -962.533,E2 -962.533} C_VEL
LIN {X 0,Y 594.282,Z 636.868,A -85,B 0,C 180,E1 -965.59,E2 -965.59} C_VEL
LIN {X 0,Y 594.273,Z 632.746,A -85,B 0,C 180,E1 -967.763,E2 -967.763} C_VEL
LIN {X 0,Y 594.279,Z 628.676,A -85,B 0,C 180,E1 -969.943,E2 -969.943} C_VEL
LIN {X 0,Y 594.313,Z 624.727,A -85,B 0,C 180,E1 -972.094,E2 -972.094} C_VEL
LIN {X 0,Y 594.293,Z 620.907,A -85,B 0,C 180,E1 -974.217,E2 -974.217} C_VEL
LIN {X 0,Y 594.324,Z 616.024,A -85,B 0,C 180,E1 -977.016,E2 -977.016} C_VEL
LIN {X 0,Y 594.359,Z 611.315,A -85,B 0,C 180,E1 -979.783,E2 -979.783} C_VEL
LIN {X 0,Y 594.325,Z 610.456,A -85,B 0,C 180,E1 -980.47,E2 -980.47} C_VEL
LIN {X 0,Y 594.4,Z 610.448,A -85,B 0,C 180,E1 -982.527,E2 -982.527} C_VEL
LIN {X 0,Y 594.387,Z 610.447,A -85,B 0,C 180,E1 -985.252,E2 -985.252} C_VEL
LIN {X 0,Y 594.406,Z 610.444,A -85,B 0,C 180,E1 -987.967,E2 -987.967} C_VEL
LIN {X 0,Y 594.427,Z 610.444,A -85,B 0,C 180,E1 -990.677,E2 -990.677} C_VEL
LIN {X 0,Y 594.386,Z 610.448,A -85,B 0,C 180,E1 -993.389,E2 -993.389} C_VEL
LIN {X 0,Y 594.376,Z 610.448,A -85,B 0,C 180,E1 -996.109,E2 -996.109} C_VEL
LIN {X 0,Y 594.367,Z 610.451,A -85,B 0,C 180,E1 -998.842,E2 -998.842} C_VEL
LIN {X 0,Y 594.288,Z 610.617,A -85,B 0,C 180,E1 -999.272,E2 -999.272} C_VEL
LIN {X 0,Y 594.313,Z 615.053,A -85,B 0,C 180,E1 -1001.597,E2 -1001.597} C_VEL
LIN {X 0,Y 594.317,Z 620.026,A -85,B 0,C 180,E1 -1004.378,E2 -1004.378} C_VEL
LIN {X 0,Y 594.299,Z 625.091,A -85,B 0,C 180,E1 -1007.196,E2 -1007.196} C_VEL
LIN {X 0,Y 594.292,Z 629.026,A -85,B 0,C 180,E1 -1009.337,E2 -1009.337} C_VEL
LIN {X 0,Y 594.287,Z 633.082,A -85,B 0,C 180,E1 -1011.506,E2 -1011.506} C_VEL
LIN {X 0,Y 594.252,Z 637.27,A -85,B 0,C 180,E1 -1013.709,E2 -1013.709} C_VEL
LIN {X 0,Y 594.26,Z 643.054,A -85,B 0,C 180,E1 -1016.705,E2 -1016.705} C_VEL
LIN {X 0,Y 594.249,Z 647.562,A -85,B 0,C 180,E1 -1019.005,E2 -1019.005} C_VEL
LIN {X 0,Y 594.249,Z 653.68,A -85,B 0,C 180,E1 -1022.032,E2 -1022.032} C_VEL
LIN {X 0,Y 594.672,Z 659.009,A -85,B 0,C 180,E1 -1022.141,E2 -1022.141} C_VEL
LIN {X 0,Y 594.612,Z 671.727,A -85,B 0,C 180,E1 -1022.482,E2 -1022.482} C_VEL
LIN {X 0,Y 594.561,Z 683.713,A -85,B 0,C 180,E1 -1022.938,E2 -1022.938} C_VEL
LIN {X 0,Y 594.455,Z 694.111,A -85,B 0,C 180,E1 -1023.451,E2 -1023.451} C_VEL
LIN {X 0,Y 594.448,Z 705.345,A -85,B 0,C 180,E1 -1024.147,E2 -1024.147} C_VEL
LIN {X 0,Y 594.38,Z 716.155,A -85,B 0,C 180,E1 -1024.992,E2 -1024.992} C_VEL
LIN {X 0,Y 594.353,Z 724.821,A -85,B 0,C 180,E1 -1025.825,E2 -1025.825} C_VEL
LIN {X 0,Y 594.31,Z 732.809,A -85,B 0,C 180,E1 -1026.757,E2 -1026.757} C_VEL
LIN {X 0,Y 594.284,Z 739.715,A -85,B 0,C 180,E1 -1027.746,E2 -1027.746} C_VEL
LIN {X 0,Y 594.266,Z 745.691,A -85,B 0,C 180,E1 -1028.814,E2 -1028.814} C_VEL
LIN {X 0,Y 594.256,Z 749.876,A -85,B 0,C 180,E1 -1029.76,E2 -1029.76} C_VEL
LIN {X 0,Y 594.23,Z 753.417,A -85,B 0,C 180,E1 -1030.805,E2 -1030.805} C_VEL
LIN {X 0,Y 594.247,Z 755.876,A -85,B 0,C 180,E1 -1031.833,E2 -1031.833} C_VEL
LIN {X 0,Y 594.248,Z 757.355,A -85,B 0,C 180,E1 -1032.84,E2 -1032.84} C_VEL
LIN {X 0,Y 594.229,Z 757.959,A -85,B 0,C 180,E1 -1034.25,E2 -1034.25} C_VEL
LIN {X 0,Y 594.229,Z 757.409,A -85,B 0,C 180,E1 -1035.204,E2 -1035.204} C_VEL
LIN {X 0,Y 594.234,Z 756.044,A -85,B 0,C 180,E1 -1036.173,E2 -1036.173} C_VEL
LIN {X 0,Y 594.25,Z 753.765,A -85,B 0,C 180,E1 -1037.159,E2 -1037.159} C_VEL
LIN {X 0,Y 594.246,Z 749.067,A -85,B 0,C 180,E1 -1038.524,E2 -1038.524} C_VEL
LIN {X 0,Y 594.284,Z 743.781,A -85,B 0,C 180,E1 -1039.641,E2 -1039.641} C_VEL
LIN {X 0,Y 594.31,Z 737.044,A -85,B 0,C 180,E1 -1040.753,E2 -1040.753} C_VEL
LIN {X 0,Y 594.327,Z 730.033,A -85,B 0,C 180,E1 -1041.681,E2 -1041.681} C_VEL
LIN {X 0,Y 594.39,Z 722.216,A -85,B 0,C 180,E1 -1042.534,E2 -1042.534} C_VEL
LIN {X 0,Y 594.433,Z 712.263,A -85,B 0,C 180,E1 -1043.422,E2 -1043.422} C_VEL
LIN {X 0,Y 594.435,Z 701.806,A -85,B 0,C 180,E1 -1044.18,E2 -1044.18} C_VEL
LIN {X 0,Y 594.538,Z 690.935,A -85,B 0,C 180,E1 -1044.811,E2 -1044.811} C_VEL
LIN {X 0,Y 594.559,Z 678.198,A -85,B 0,C 180,E1 -1045.38,E2 -1045.38} C_VEL
LIN {X 0,Y 594.646,Z 665.51,A -85,B 0,C 180,E1 -1045.792,E2 -1045.792} C_VEL
LIN {X 0,Y 594.513,Z 655.493,A -85,B 0,C 180,E1 -1046.02,E2 -1046.02} C_VEL
LIN {X 0,Y 594.253,Z 653.525,A -85,B 0,C 180,E1 -1046.079,E2 -1046.079} C_VEL
LIN {X 0,Y 594.243,Z 648.436,A -85,B 0,C 180,E1 -1048.642,E2 -1048.642} C_VEL
LIN {X 0,Y 594.253,Z 643.681,A -85,B 0,C 180,E1 -1051.064,E2 -1051.064} C_VEL
LIN {X 0,Y 594.258,Z 639.355,A -85,B 0,C 180,E1 -1053.294,E2 -1053.294} C_VEL
LIN {X 0,Y 594.253,Z 633.639,A -85,B 0,C 180,E1 -1056.29,E2 -1056.29} C_VEL
LIN {X 0,Y 594.308,Z 628.382,A -85,B 0,C 180,E1 -1059.1,E2 -1059.1} C_VEL
LIN {X 0,Y 594.318,Z 624.206,A -85,B 0,C 180,E1 -1061.38,E2 -1061.38} C_VEL
LIN {X 0,Y 594.327,Z 620.378,A -85,B 0,C 180,E1 -1063.513,E2 -1063.513} C_VEL
LIN {X 0,Y 594.335,Z 615.323,A -85,B 0,C 180,E1 -1066.32,E2 -1066.32} C_VEL
LIN {X 0,Y 594.327,Z 610.458,A -85,B 0,C 180,E1 -1068.78,E2 -1068.78} C_VEL
LIN {X 0,Y 594.4,Z 610.448,A -85,B 0,C 180,E1 -1071.158,E2 -1071.158} C_VEL
LIN {X 0,Y 594.377,Z 610.45,A -85,B 0,C 180,E1 -1073.891,E2 -1073.891} C_VEL
LIN {X 0,Y 594.384,Z 610.448,A -85,B 0,C 180,E1 -1076.611,E2 -1076.611} C_VEL
LIN {X 0,Y 594.428,Z 610.445,A -85,B 0,C 180,E1 -1079.323,E2 -1079.323} C_VEL
LIN {X 0,Y 594.388,Z 610.448,A -85,B 0,C 180,E1 -1082.033,E2 -1082.033} C_VEL
LIN {X 0,Y 594.398,Z 610.446,A -85,B 0,C 180,E1 -1084.748,E2 -1084.748} C_VEL
LIN {X 0,Y 594.417,Z 610.446,A -85,B 0,C 180,E1 -1087.473,E2 -1087.473} C_VEL
LIN {X 0,Y 594.39,Z 610.447,A -85,B 0,C 180,E1 -1090.216,E2 -1090.216} C_VEL
LIN {X 0,Y 594.372,Z 610.45,A -85,B 0,C 180,E1 -1092.983,E2 -1092.983} C_VEL
LIN {X 0,Y 594.369,Z 610.452,A -85,B 0,C 180,E1 -1095.781,E2 -1095.781} C_VEL
LIN {X 0,Y 594.383,Z 610.449,A -85,B 0,C 180,E1 -1098.618,E2 -1098.618} C_VEL
LIN {X 0,Y 594.369,Z 610.45,A -85,B 0,C 180,E1 -1101.503,E2 -1101.503} C_VEL
LIN {X 0,Y 594.386,Z 610.448,A -85,B 0,C 180,E1 -1104.446,E2 -1104.446} C_VEL
LIN {X 0,Y 594.387,Z 610.448,A -85,B 0,C 180,E1 -1106.699,E2 -1106.699} C_VEL
LIN {X 0,Y 594.378,Z 610.45,A -85,B 0,C 180,E1 -1108.999,E2 -1108.999} C_VEL
LIN {X 0,Y 594.392,Z 610.447,A -85,B 0,C 180,E1 -1111.646,E2 -1111.646} C_VEL
LIN {X 0,Y 594.378,Z 610.449,A -85,B 0,C 180,E1 -1114.58,E2 -1114.58} C_VEL
LIN {X 0,Y 594.382,Z 610.449,A -85,B 0,C 180,E1 -1117.087,E2 -1117.087} C_VEL
LIN {X 0,Y 594.375,Z 610.449,A -85,B 0,C 180,E1 -1119.775,E2 -1119.775} C_VEL
LIN {X 0,Y 594.365,Z 610.452,A -85,B 0,C 180,E1 -1122.376,E2 -1122.376} C_VEL
LIN {X 0,Y 594.362,Z 610.451,A -85,B 0,C 180,E1 -1125.192,E2 -1125.192} C_VEL
LIN {X 0,Y 594.381,Z 610.448,A -85,B 0,C 180,E1 -1128.152,E2 -1128.152} C_VEL
LIN {X 0,Y 594.379,Z 610.449,A -85,B 0,C 180,E1 -1131.195,E2 -1131.195} C_VEL
LIN {X 0,Y 594.395,Z 610.448,A -85,B 0,C 180,E1 -1134.113,E2 -1134.113} C_VEL
LIN {X 0,Y 594.537,Z 615.014,A -85,B 0,C 180,E1 -1135.84,E2 -1135.84} C_VEL
LIN {X 0,Y 594.412,Z 622.849,A -85,B 0,C 180,E1 -1138.653,E2 -1138.653} C_VEL
LIN {X 0,Y 594.439,Z 630.685,A -85,B 0,C 180,E1 -1141.407,E2 -1141.407} C_VEL
LIN {X 0,Y 594.396,Z 638.432,A -85,B 0,C 180,E1 -1144.057,E2 -1144.057} C_VEL
LIN {X 0,Y 594.353,Z 646.223,A -85,B 0,C 180,E1 -1146.664,E2 -1146.664} C_VEL
LIN {X 0,Y 594.361,Z 655.127,A -85,B 0,C 180,E1 -1149.585,E2 -1149.585} C_VEL
LIN {X 0,Y 594.319,Z 664.032,A -85,B 0,C 180,E1 -1152.45,E2 -1152.45} C_VEL
LIN {X 0,Y 594.311,Z 672.936,A -85,B 0,C 180,E1 -1155.271,E2 -1155.271} C_VEL
LIN {X 0,Y 594.294,Z 681.493,A -85,B 0,C 180,E1 -1157.948,E2 -1157.948} C_VEL
LIN {X 0,Y 594.678,Z 686.249,A -85,B 0,C 180,E1 -1158.043,E2 -1158.043} C_VEL
LIN {X 0,Y 594.612,Z 699.509,A -85,B 0,C 180,E1 -1158.366,E2 -1158.366} C_VEL
LIN {X 0,Y 594.545,Z 711.503,A -85,B 0,C 180,E1 -1158.795,E2 -1158.795} C_VEL
LIN {X 0,Y 594.5,Z 723.215,A -85,B 0,C 180,E1 -1159.356,E2 -1159.356} C_VEL
LIN {X 0,Y 594.462,Z 734.482,A -85,B 0,C 180,E1 -1160.044,E2 -1160.044} C_VEL
LIN {X 0,Y 594.406,Z 744.651,A -85,B 0,C 180,E1 -1160.816,E2 -1160.816} C_VEL
LIN {X 0,Y 594.372,Z 753.791,A -85,B 0,C 180,E1 -1161.672,E2 -1161.672} C_VEL
LIN {X 0,Y 594.316,Z 762.694,A -85,B 0,C 180,E1 -1162.697,E2 -1162.697} C_VEL
LIN {X 0,Y 594.281,Z 769.167,A -85,B 0,C 180,E1 -1163.614,E2 -1163.614} C_VEL
LIN {X 0,Y 594.289,Z 774.682,A -85,B 0,C 180,E1 -1164.572,E2 -1164.572} C_VEL
LIN {X 0,Y 594.27,Z 779.372,A -85,B 0,C 180,E1 -1165.592,E2 -1165.592} C_VEL
LIN {X 0,Y 594.267,Z 782.957,A -85,B 0,C 180,E1 -1166.61,E2 -1166.61} C_VEL
LIN {X 0,Y 594.225,Z 784.81,A -85,B 0,C 180,E1 -1167.289,E2 -1167.289} C_VEL
LIN {X 0,Y 594.241,Z 786.202,A -85,B 0,C 180,E1 -1167.967,E2 -1167.967} C_VEL
LIN {X 0,Y 594.239,Z 787.784,A -85,B 0,C 180,E1 -1169.323,E2 -1169.323} C_VEL
LIN {X 0,Y 594.236,Z 788,A -85,B 0,C 180,E1 -1170,E2 -1170} C_VEL
LIN {X 0,Y 594.247,Z 787.184,A -85,B 0,C 180,E1 -1171.356,E2 -1171.356} C_VEL
LIN {X 0,Y 594.241,Z 786.202,A -85,B 0,C 180,E1 -1172.034,E2 -1172.034} C_VEL
LIN {X 0,Y 594.226,Z 784.809,A -85,B 0,C 180,E1 -1172.712,E2 -1172.712} C_VEL
LIN {X 0,Y 594.289,Z 781.895,A -85,B 0,C 180,E1 -1173.73,E2 -1173.73} C_VEL
LIN {X 0,Y 594.241,Z 777.949,A -85,B 0,C 180,E1 -1174.749,E2 -1174.749} C_VEL
LIN {X 0,Y 594.304,Z 771.876,A -85,B 0,C 180,E1 -1175.94,E2 -1175.94} C_VEL
LIN {X 0,Y 594.308,Z 765.234,A -85,B 0,C 180,E1 -1176.962,E2 -1176.962} C_VEL
LIN {X 0,Y 594.359,Z 756.987,A -85,B 0,C 180,E1 -1177.987,E2 -1177.987} C_VEL
LIN {X 0,Y 594.382,Z 748.534,A -85,B 0,C 180,E1 -1178.842,E2 -1178.842} C_VEL
LIN {X 0,Y 594.435,Z 738.09,A -85,B 0,C 180,E1 -1179.7,E2 -1179.7} C_VEL
LIN {X 0,Y 594.482,Z 727.754,A -85,B 0,C 180,E1 -1180.387,E2 -1180.387} C_VEL
LIN {X 0,Y 594.509,Z 715.683,A -85,B 0,C 180,E1 -1181.023,E2 -1181.023} C_VEL
LIN {X 0,Y 594.557,Z 703.472,A -85,B 0,C 180,E1 -1181.506,E2 -1181.506} C_VEL
LIN {X 0,Y 594.633,Z 690.428,A -85,B 0,C 180,E1 -1181.872,E2 -1181.872} C_VEL
LIN {X 0,Y 594.433,Z 682.598,A -85,B 0,C 180,E1 -1182.028,E2 -1182.028} C_VEL
LIN {X 0,Y 594.3,Z 681.421,A -85,B 0,C 180,E1 -1182.074,E2 -1182.074} C_VEL
LIN {X 0,Y 594.289,Z 671.821,A -85,B 0,C 180,E1 -1185.08,E2 -1185.08} C_VEL
LIN {X 0,Y 594.328,Z 662.917,A -85,B 0,C 180,E1 -1187.906,E2 -1187.906} C_VEL
LIN {X 0,Y 594.354,Z 654.013,A -85,B 0,C 180,E1 -1190.778,E2 -1190.778} C_VEL
LIN {X 0,Y 594.382,Z 645.108,A -85,B 0,C 180,E1 -1193.705,E2 -1193.705} C_VEL
LIN {X 0,Y 594.39,Z 638.195,A -85,B 0,C 180,E1 -1196.023,E2 -1196.023} C_VEL
LIN {X 0,Y 594.441,Z 630.684,A -85,B 0,C 180,E1 -1198.593,E2 -1198.593} C_VEL
LIN {X 0,Y 594.414,Z 622.847,A -85,B 0,C 180,E1 -1201.348,E2 -1201.348} C_VEL
LIN {X 0,Y 594.449,Z 616.092,A -85,B 0,C 180,E1 -1203.757,E2 -1203.757} C_VEL
LIN {X 0,Y 594.546,Z 611.683,A -85,B 0,C 180,E1 -1205.396,E2 -1205.396} C_VEL
LIN {X 0,Y 594.374,Z 610.451,A -85,B 0,C 180,E1 -1205.929,E2 -1205.929} C_VEL
LIN {X 0,Y 594.382,Z 610.448,A -85,B 0,C 180,E1 -1208.805,E2 -1208.805} C_VEL
LIN {X 0,Y 594.385,Z 610.448,A -85,B 0,C 180,E1 -1211.848,E2 -1211.848} C_VEL
LIN {X 0,Y 594.385,Z 610.451,A -85,B 0,C 180,E1 -1214.236,E2 -1214.236} C_VEL
LIN {X 0,Y 594.362,Z 610.452,A -85,B 0,C 180,E1 -1217.148,E2 -1217.148} C_VEL
LIN {X 0,Y 594.369,Z 610.452,A -85,B 0,C 180,E1 -1219.433,E2 -1219.433} C_VEL
LIN {X 0,Y 594.39,Z 610.45,A -85,B 0,C 180,E1 -1222.392,E2 -1222.392} C_VEL
LIN {X 0,Y 594.396,Z 610.449,A -85,B 0,C 180,E1 -1225.421,E2 -1225.421} C_VEL
LIN {X 0,Y 594.393,Z 610.449,A -85,B 0,C 180,E1 -1228.355,E2 -1228.355} C_VEL
LIN {X 0,Y 594.385,Z 610.448,A -85,B 0,C 180,E1 -1231.042,E2 -1231.042} C_VEL
LIN {X 0,Y 594.388,Z 610.447,A -85,B 0,C 180,E1 -1233.977,E2 -1233.977} C_VEL
LIN {X 0,Y 594.389,Z 610.448,A -85,B 0,C 180,E1 -1236.296,E2 -1236.296} C_VEL
LIN {X 0,Y 594.408,Z 610.445,A -85,B 0,C 180,E1 -1239.225,E2 -1239.225} C_VEL
LIN {X 0,Y 594.355,Z 610.452,A -85,B 0,C 180,E1 -1242.095,E2 -1242.095} C_VEL
LIN {X 0,Y 594.37,Z 610.45,A -85,B 0,C 180,E1 -1244.219,E2 -1244.219} C_VEL
LIN {X 0,Y 594.371,Z 610.45,A -85,B 0,C 180,E1 -1247.017,E2 -1247.017} C_VEL
LIN {X 0,Y 594.39,Z 610.449,A -85,B 0,C 180,E1 -1249.784,E2 -1249.784} C_VEL
LIN {X 0,Y 594.405,Z 610.446,A -85,B 0,C 180,E1 -1252.527,E2 -1252.527} C_VEL
LIN {X 0,Y 594.395,Z 610.447,A -85,B 0,C 180,E1 -1255.252,E2 -1255.252} C_VEL
LIN {X 0,Y 594.392,Z 610.448,A -85,B 0,C 180,E1 -1257.967,E2 -1257.967} C_VEL
LIN {X 0,Y 594.429,Z 610.444,A -85,B 0,C 180,E1 -1260.677,E2 -1260.677} C_VEL
LIN {X 0,Y 594.384,Z 610.448,A -85,B 0,C 180,E1 -1263.389,E2 -1263.389} C_VEL
LIN {X 0,Y 594.376,Z 610.45,A -85,B 0,C 180,E1 -1266.109,E2 -1266.109} C_VEL
LIN {X 0,Y 594.401,Z 610.449,A -85,B 0,C 180,E1 -1268.842,E2 -1268.842} C_VEL
LIN {X 0,Y 594.353,Z 610.452,A -85,B 0,C 180,E1 -1269.529,E2 -1269.529} C_VEL
LIN {X 0,Y 594.366,Z 611.221,A -85,B 0,C 180,E1 -1270.216,E2 -1270.216} C_VEL
LIN {X 0,Y 594.32,Z 615.835,A -85,B 0,C 180,E1 -1272.984,E2 -1272.984} C_VEL
LIN {X 0,Y 594.291,Z 619.776,A -85,B 0,C 180,E1 -1275.236,E2 -1275.236} C_VEL
LIN {X 0,Y 593.605,Z 620.83,A -85,B 0,C 180,E1 -1275.793,E2 -1275.793} C_VEL
LIN {X 0,Y 590.744,Z 622.705,A -85,B 0,C 180,E1 -1276.693,E2 -1276.693} C_VEL
LIN {X 0,Y 588.339,Z 624.221,A -85,B 0,C 180,E1 -1277.417,E2 -1277.417} C_VEL
LIN {X 0,Y 587.309,Z 625.318,A -85,B 0,C 180,E1 -1277.976,E2 -1277.976} C_VEL
LIN {X 0,Y 587.226,Z 625.666,A -85,B 0,C 180,E1 -1278.166,E2 -1278.166} C_VEL
LIN {X 0,Y 587.243,Z 630.899,A -85,B 0,C 180,E1 -1281.041,E2 -1281.041} C_VEL
LIN {X 0,Y 587.198,Z 635.032,A -85,B 0,C 180,E1 -1283.264,E2 -1283.264} C_VEL
LIN {X 0,Y 587.19,Z 640.748,A -85,B 0,C 180,E1 -1286.286,E2 -1286.286} C_VEL
LIN {X 0,Y 587.17,Z 646.168,A -85,B 0,C 180,E1 -1289.102,E2 -1289.102} C_VEL
LIN {X 0,Y 587.135,Z 651.439,A -85,B 0,C 180,E1 -1291.803,E2 -1291.803} C_VEL
LIN {X 0,Y 587.181,Z 653.683,A -85,B 0,C 180,E1 -1292.884,E2 -1292.884} C_VEL
LIN {X 0,Y 587.722,Z 659.297,A -85,B 0,C 180,E1 -1293.004,E2 -1293.004} C_VEL
LIN {X 0,Y 587.644,Z 671.164,A -85,B 0,C 180,E1 -1293.324,E2 -1293.324} C_VEL
LIN {X 0,Y 587.552,Z 683.52,A -85,B 0,C 180,E1 -1293.794,E2 -1293.794} C_VEL
LIN {X 0,Y 587.513,Z 694.985,A -85,B 0,C 180,E1 -1294.371,E2 -1294.371} C_VEL
LIN {X 0,Y 587.442,Z 705.646,A -85,B 0,C 180,E1 -1295.048,E2 -1295.048} C_VEL
LIN {X 0,Y 587.394,Z 716.262,A -85,B 0,C 180,E1 -1295.893,E2 -1295.893} C_VEL
LIN {X 0,Y 587.275,Z 725.075,A -85,B 0,C 180,E1 -1296.752,E2 -1296.752} C_VEL
LIN {X 0,Y 587.236,Z 733.995,A -85,B 0,C 180,E1 -1297.825,E2 -1297.825} C_VEL
LIN {X 0,Y 587.209,Z 741.249,A -85,B 0,C 180,E1 -1298.927,E2 -1298.927} C_VEL
LIN {X 0,Y 587.208,Z 746.883,A -85,B 0,C 180,E1 -1300.005,E2 -1300.005} C_VEL
LIN {X 0,Y 587.141,Z 751.566,A -85,B 0,C 180,E1 -1301.174,E2 -1301.174} C_VEL
LIN {X 0,Y 587.165,Z 754.267,A -85,B 0,C 180,E1 -1302.089,E2 -1302.089} C_VEL
LIN {X 0,Y 587.148,Z 756.385,A -85,B 0,C 180,E1 -1303.101,E2 -1303.101} C_VEL
LIN {X 0,Y 587.157,Z 757.605,A -85,B 0,C 180,E1 -1304.096,E2 -1304.096} C_VEL
LIN {X 0,Y 587.146,Z 757.998,A -85,B 0,C 180,E1 -1305.072,E2 -1305.072} C_VEL
LIN {X 0,Y 587.138,Z 757.579,A -85,B 0,C 180,E1 -1306.032,E2 -1306.032} C_VEL
LIN {X 0,Y 587.165,Z 756.399,A -85,B 0,C 180,E1 -1306.98,E2 -1306.98} C_VEL
LIN {X 0,Y 587.165,Z 753.279,A -85,B 0,C 180,E1 -1308.371,E2 -1308.371} C_VEL
LIN {X 0,Y 587.162,Z 750.032,A -85,B 0,C 180,E1 -1309.342,E2 -1309.342} C_VEL
LIN {X 0,Y 587.21,Z 745.812,A -85,B 0,C 180,E1 -1310.313,E2 -1310.313} C_VEL
LIN {X 0,Y 587.235,Z 740.479,A -85,B 0,C 180,E1 -1311.295,E2 -1311.295} C_VEL
LIN {X 0,Y 587.242,Z 733.101,A -85,B 0,C 180,E1 -1312.384,E2 -1312.384} C_VEL
LIN {X 0,Y 587.284,Z 725.414,A -85,B 0,C 180,E1 -1313.301,E2 -1313.301} C_VEL
LIN {X 0,Y 587.376,Z 716.152,A -85,B 0,C 180,E1 -1314.207,E2 -1314.207} C_VEL
LIN {X 0,Y 587.428,Z 705.617,A -85,B 0,C 180,E1 -1315.044,E2 -1315.044} C_VEL
LIN {X 0,Y 587.528,Z 693.684,A -85,B 0,C 180,E1 -1315.791,E2 -1315.791} C_VEL
LIN {X 0,Y 587.579,Z 682.01,A -85,B 0,C 180,E1 -1316.362,E2 -1316.362} C_VEL
LIN {X 0,Y 587.684,Z 670.154,A -85,B 0,C 180,E1 -1316.799,E2 -1316.799} C_VEL
LIN {X 0,Y 587.647,Z 656.665,A -85,B 0,C 180,E1 -1317.139,E2 -1317.139} C_VEL
LIN {X 0,Y 587.164,Z 653.533,A -85,B 0,C 180,E1 -1317.222,E2 -1317.222} C_VEL
LIN {X 0,Y 587.161,Z 648.44,A -85,B 0,C 180,E1 -1319.82,E2 -1319.82} C_VEL
LIN {X 0,Y 587.172,Z 643.554,A -85,B 0,C 180,E1 -1322.341,E2 -1322.341} C_VEL
LIN {X 0,Y 587.178,Z 638.032,A -85,B 0,C 180,E1 -1325.233,E2 -1325.233} C_VEL
LIN {X 0,Y 587.221,Z 633.806,A -85,B 0,C 180,E1 -1327.481,E2 -1327.481} C_VEL
LIN {X 0,Y 587.202,Z 629.724,A -85,B 0,C 180,E1 -1329.69,E2 -1329.69} C_VEL
LIN {X 0,Y 587.233,Z 625.762,A -85,B 0,C 180,E1 -1331.87,E2 -1331.87} C_VEL
LIN {X 0,Y 587.236,Z 621.927,A -85,B 0,C 180,E1 -1334.022,E2 -1334.022} C_VEL
LIN {X 0,Y 587.268,Z 617.109,A -85,B 0,C 180,E1 -1336.857,E2 -1336.857} C_VEL
LIN {X 0,Y 587.318,Z 612.334,A -85,B 0,C 180,E1 -1339.659,E2 -1339.659} C_VEL
LIN {X 0,Y 587.263,Z 611.336,A -85,B 0,C 180,E1 -1340.355,E2 -1340.355} C_VEL
LIN {X 0,Y 587.373,Z 611.322,A -85,B 0,C 180,E1 -1342.437,E2 -1342.437} C_VEL
LIN {X 0,Y 587.359,Z 611.323,A -85,B 0,C 180,E1 -1345.195,E2 -1345.195} C_VEL
LIN {X 0,Y 587.376,Z 611.32,A -85,B 0,C 180,E1 -1347.943,E2 -1347.943} C_VEL
LIN {X 0,Y 587.398,Z 611.32,A -85,B 0,C 180,E1 -1350.685,E2 -1350.685} C_VEL
LIN {X 0,Y 587.338,Z 611.325,A -85,B 0,C 180,E1 -1353.43,E2 -1353.43} C_VEL
LIN {X 0,Y 587.332,Z 611.325,A -85,B 0,C 180,E1 -1356.182,E2 -1356.182} C_VEL
LIN {X 0,Y 587.365,Z 611.322,A -85,B 0,C 180,E1 -1358.255,E2 -1358.255} C_VEL
LIN {X 0,Y 587.229,Z 611.445,A -85,B 0,C 180,E1 -1359.384,E2 -1359.384} C_VEL
LIN {X 0,Y 587.246,Z 615.914,A -85,B 0,C 180,E1 -1361.738,E2 -1361.738} C_VEL
LIN {X 0,Y 587.257,Z 621.023,A -85,B 0,C 180,E1 -1364.555,E2 -1364.555} C_VEL
LIN {X 0,Y 587.222,Z 626.105,A -85,B 0,C 180,E1 -1367.409,E2 -1367.409} C_VEL
LIN {X 0,Y 587.213,Z 630.052,A -85,B 0,C 180,E1 -1369.579,E2 -1369.579} C_VEL
LIN {X 0,Y 587.191,Z 634.126,A -85,B 0,C 180,E1 -1371.779,E2 -1371.779} C_VEL
LIN {X 0,Y 587.194,Z 639.337,A -85,B 0,C 180,E1 -1374.545,E2 -1374.545} C_VEL
LIN {X 0,Y 587.16,Z 644.143,A -85,B 0,C 180,E1 -1377.054,E2 -1377.054} C_VEL
LIN {X 0,Y 587.152,Z 648.674,A -85,B 0,C 180,E1 -1379.39,E2 -1379.39} C_VEL
LIN {X 0,Y 587.16,Z 653.548,A -85,B 0,C 180,E1 -1381.875,E2 -1381.875} C_VEL
LIN {X 0,Y 587.734,Z 658.886,A -85,B 0,C 180,E1 -1381.995,E2 -1381.995} C_VEL
LIN {X 0,Y 587.66,Z 671.474,A -85,B 0,C 180,E1 -1382.335,E2 -1382.335} C_VEL
LIN {X 0,Y 587.586,Z 683.466,A -85,B 0,C 180,E1 -1382.794,E2 -1382.794} C_VEL
LIN {X 0,Y 587.461,Z 695.267,A -85,B 0,C 180,E1 -1383.388,E2 -1383.388} C_VEL
LIN {X 0,Y 587.432,Z 706.527,A -85,B 0,C 180,E1 -1384.111,E2 -1384.111} C_VEL
LIN {X 0,Y 587.346,Z 717.007,A -85,B 0,C 180,E1 -1384.959,E2 -1384.959} C_VEL
LIN {X 0,Y 587.282,Z 726.422,A -85,B 0,C 180,E1 -1385.9,E2 -1385.9} C_VEL
LIN {X 0,Y 587.231,Z 733.455,A -85,B 0,C 180,E1 -1386.755,E2 -1386.755} C_VEL
LIN {X 0,Y 587.199,Z 740.632,A -85,B 0,C 180,E1 -1387.82,E2 -1387.82} C_VEL
LIN {X 0,Y 587.185,Z 746.506,A -85,B 0,C 180,E1 -1388.923,E2 -1388.923} C_VEL
LIN {X 0,Y 587.184,Z 750.954,A -85,B 0,C 180,E1 -1390.002,E2 -1390.002} C_VEL
LIN {X 0,Y 587.126,Z 754.49,A -85,B 0,C 180,E1 -1391.174,E2 -1391.174} C_VEL
LIN {X 0,Y 587.162,Z 756.367,A -85,B 0,C 180,E1 -1392.089,E2 -1392.089} C_VEL
LIN {X 0,Y 587.146,Z 757.61,A -85,B 0,C 180,E1 -1393.1,E2 -1393.1} C_VEL
LIN {X 0,Y 587.154,Z 757.995,A -85,B 0,C 180,E1 -1394.096,E2 -1394.096} C_VEL
LIN {X 0,Y 587.151,Z 757.553,A -85,B 0,C 180,E1 -1395.072,E2 -1395.072} C_VEL
LIN {X 0,Y 587.134,Z 756.319,A -85,B 0,C 180,E1 -1396.031,E2 -1396.031} C_VEL
LIN {X 0,Y 587.167,Z 754.325,A -85,B 0,C 180,E1 -1396.98,E2 -1396.98} C_VEL
LIN {X 0,Y 587.191,Z 751.578,A -85,B 0,C 180,E1 -1397.913,E2 -1397.913} C_VEL
LIN {X 0,Y 587.183,Z 747.555,A -85,B 0,C 180,E1 -1398.941,E2 -1398.941} C_VEL
LIN {X 0,Y 587.208,Z 742.248,A -85,B 0,C 180,E1 -1399.994,E2 -1399.994} C_VEL
LIN {X 0,Y 587.264,Z 735.417,A -85,B 0,C 180,E1 -1401.066,E2 -1401.066} C_VEL
LIN {X 0,Y 587.3,Z 727.701,A -85,B 0,C 180,E1 -1402.045,E2 -1402.045} C_VEL
LIN {X 0,Y 587.35,Z 719.171,A -85,B 0,C 180,E1 -1402.931,E2 -1402.931} C_VEL
LIN {X 0,Y 587.422,Z 709.036,A -85,B 0,C 180,E1 -1403.791,E2 -1403.791} C_VEL
LIN {X 0,Y 587.472,Z 697.179,A -85,B 0,C 180,E1 -1404.593,E2 -1404.593} C_VEL
LIN {X 0,Y 587.577,Z 685.441,A -85,B 0,C 180,E1 -1405.208,E2 -1405.208} C_VEL
LIN {X 0,Y 587.63,Z 673.701,A -85,B 0,C 180,E1 -1405.68,E2 -1405.68} C_VEL
LIN {X 0,Y 587.703,Z 660.361,A -85,B 0,C 180,E1 -1406.061,E2 -1406.061} C_VEL
LIN {X 0,Y 587.4,Z 655.338,A -85,B 0,C 180,E1 -1406.17,E2 -1406.17} C_VEL
LIN {X 0,Y 587.179,Z 653.536,A -85,B 0,C 180,E1 -1406.22,E2 -1406.22} C_VEL
LIN {X 0,Y 587.145,Z 648.046,A -85,B 0,C 180,E1 -1409.022,E2 -1409.022} C_VEL
LIN {X 0,Y 587.151,Z 643.454,A -85,B 0,C 180,E1 -1411.394,E2 -1411.394} C_VEL
LIN {X 0,Y 587.198,Z 638.757,A -85,B 0,C 180,E1 -1413.85,E2 -1413.85} C_VEL
LIN {X 0,Y 587.186,Z 633.336,A -85,B 0,C 180,E1 -1416.735,E2 -1416.735} C_VEL
LIN {X 0,Y 587.231,Z 629.18,A -85,B 0,C 180,E1 -1418.987,E2 -1418.987} C_VEL
LIN {X 0,Y 587.235,Z 623.97,A -85,B 0,C 180,E1 -1421.87,E2 -1421.87} C_VEL
LIN {X 0,Y 587.242,Z 620.171,A -85,B 0,C 180,E1 -1424.022,E2 -1424.022} C_VEL
LIN {X 0,Y 587.259,Z 616.15,A -85,B 0,C 180,E1 -1426.152,E2 -1426.152} C_VEL
LIN {X 0,Y 587.24,Z 611.34,A -85,B 0,C 180,E1 -1428.568,E2 -1428.568} C_VEL
LIN {X 0,Y 587.345,Z 611.328,A -85,B 0,C 180,E1 -1431.051,E2 -1431.051} C_VEL
LIN {X 0,Y 587.373,Z 611.323,A -85,B 0,C 180,E1 -1433.263,E2 -1433.263} C_VEL
LIN {X 0,Y 587.319,Z 611.328,A -85,B 0,C 180,E1 -1435.883,E2 -1435.883} C_VEL
LIN {X 0,Y 587.365,Z 611.323,A -85,B 0,C 180,E1 -1437.943,E2 -1437.943} C_VEL
LIN {X 0,Y 587.393,Z 611.319,A -85,B 0,C 180,E1 -1440.686,E2 -1440.686} C_VEL
LIN {X 0,Y 587.338,Z 611.328,A -85,B 0,C 180,E1 -1443.43,E2 -1443.43} C_VEL
LIN {X 0,Y 587.36,Z 611.325,A -85,B 0,C 180,E1 -1445.493,E2 -1445.493} C_VEL
LIN {X 0,Y 587.368,Z 611.322,A -85,B 0,C 180,E1 -1448.255,E2 -1448.255} C_VEL
LIN {X 0,Y 587.359,Z 611.323,A -85,B 0,C 180,E1 -1451.141,E2 -1451.141} C_VEL
LIN {X 0,Y 587.362,Z 611.322,A -85,B 0,C 180,E1 -1454.261,E2 -1454.261} C_VEL
LIN {X 0,Y 587.357,Z 611.323,A -85,B 0,C 180,E1 -1457.406,E2 -1457.406} C_VEL
LIN {X 0,Y 587.328,Z 611.327,A -85,B 0,C 180,E1 -1460.305,E2 -1460.305} C_VEL
LIN {X 0,Y 587.322,Z 611.328,A -85,B 0,C 180,E1 -1463.259,E2 -1463.259} C_VEL
LIN {X 0,Y 587.337,Z 611.326,A -85,B 0,C 180,E1 -1465.517,E2 -1465.517} C_VEL
LIN {X 0,Y 587.346,Z 611.325,A -85,B 0,C 180,E1 -1467.818,E2 -1467.818} C_VEL
LIN {X 0,Y 587.349,Z 611.324,A -85,B 0,C 180,E1 -1470.513,E2 -1470.513} C_VEL
LIN {X 0,Y 587.335,Z 611.327,A -85,B 0,C 180,E1 -1473.397,E2 -1473.397} C_VEL
LIN {X 0,Y 587.317,Z 611.328,A -85,B 0,C 180,E1 -1475.898,E2 -1475.898} C_VEL
LIN {X 0,Y 587.329,Z 611.328,A -85,B 0,C 180,E1 -1478.48,E2 -1478.48} C_VEL
LIN {X 0,Y 587.335,Z 611.326,A -85,B 0,C 180,E1 -1481.157,E2 -1481.157} C_VEL
LIN {X 0,Y 587.31,Z 611.329,A -85,B 0,C 180,E1 -1484.112,E2 -1484.112} C_VEL
LIN {X 0,Y 587.315,Z 611.329,A -85,B 0,C 180,E1 -1486.994,E2 -1486.994} C_VEL
LIN {X 0,Y 587.313,Z 611.331,A -85,B 0,C 180,E1 -1489.746,E2 -1489.746} C_VEL
LIN {X 0,Y 587.345,Z 611.325,A -85,B 0,C 180,E1 -1492.393,E2 -1492.393} C_VEL
LIN {X 0,Y 587.369,Z 611.425,A -85,B 0,C 180,E1 -1494,E2 -1494} C_VEL
LIN {X 0,Y 587.536,Z 616.1,A -85,B 0,C 180,E1 -1495.792,E2 -1495.792} C_VEL
LIN {X 0,Y 587.441,Z 622.845,A -85,B 0,C 180,E1 -1498.238,E2 -1498.238} C_VEL
LIN {X 0,Y 587.403,Z 629.527,A -85,B 0,C 180,E1 -1500.624,E2 -1500.624} C_VEL
LIN {X 0,Y 587.378,Z 637.319,A -85,B 0,C 180,E1 -1503.341,E2 -1503.341} C_VEL
LIN {X 0,Y 587.357,Z 645.11,A -85,B 0,C 180,E1 -1505.995,E2 -1505.995} C_VEL
LIN {X 0,Y 587.297,Z 654.045,A -85,B 0,C 180,E1 -1508.972,E2 -1508.972} C_VEL
LIN {X 0,Y 587.264,Z 662.919,A -85,B 0,C 180,E1 -1511.872,E2 -1511.872} C_VEL
LIN {X 0,Y 587.245,Z 670.71,A -85,B 0,C 180,E1 -1514.379,E2 -1514.379} C_VEL
LIN {X 0,Y 587.208,Z 679.615,A -85,B 0,C 180,E1 -1517.208,E2 -1517.208} C_VEL
LIN {X 0,Y 587.196,Z 681.493,A -85,B 0,C 180,E1 -1517.8,E2 -1517.8} C_VEL
LIN {X 0,Y 587.758,Z 686.249,A -85,B 0,C 180,E1 -1517.9,E2 -1517.9} C_VEL
LIN {X 0,Y 587.678,Z 699.509,A -85,B 0,C 180,E1 -1518.227,E2 -1518.227} C_VEL
LIN {X 0,Y 587.583,Z 711.282,A -85,B 0,C 180,E1 -1518.651,E2 -1518.651} C_VEL
LIN {X 0,Y 587.52,Z 723.216,A -85,B 0,C 180,E1 -1519.228,E2 -1519.228} C_VEL
LIN {X 0,Y 587.459,Z 734.483,A -85,B 0,C 180,E1 -1519.924,E2 -1519.924} C_VEL
LIN {X 0,Y 587.384,Z 744.651,A -85,B 0,C 180,E1 -1520.705,E2 -1520.705} C_VEL
LIN {X 0,Y 587.339,Z 753.79,A -85,B 0,C 180,E1 -1521.571,E2 -1521.571} C_VEL
LIN {X 0,Y 587.258,Z 762.693,A -85,B 0,C 180,E1 -1522.609,E2 -1522.609} C_VEL
LIN {X 0,Y 587.196,Z 769.744,A -85,B 0,C 180,E1 -1523.627,E2 -1523.627} C_VEL
LIN {X 0,Y 587.211,Z 774.682,A -85,B 0,C 180,E1 -1524.506,E2 -1524.506} C_VEL
LIN {X 0,Y 587.189,Z 779.373,A -85,B 0,C 180,E1 -1525.538,E2 -1525.538} C_VEL
LIN {X 0,Y 587.193,Z 782.957,A -85,B 0,C 180,E1 -1526.569,E2 -1526.569} C_VEL
LIN {X 0,Y 587.132,Z 784.809,A -85,B 0,C 180,E1 -1527.256,E2 -1527.256} C_VEL
LIN {X 0,Y 587.14,Z 786.201,A -85,B 0,C 180,E1 -1527.942,E2 -1527.942} C_VEL
LIN {X 0,Y 587.14,Z 787.784,A -85,B 0,C 180,E1 -1529.314,E2 -1529.314} C_VEL
LIN {X 0,Y 587.137,Z 788,A -85,B 0,C 180,E1 -1530,E2 -1530} C_VEL
LIN {X 0,Y 587.147,Z 787.185,A -85,B 0,C 180,E1 -1531.372,E2 -1531.372} C_VEL
LIN {X 0,Y 587.14,Z 786.201,A -85,B 0,C 180,E1 -1532.058,E2 -1532.058} C_VEL
LIN {X 0,Y 587.132,Z 784.809,A -85,B 0,C 180,E1 -1532.745,E2 -1532.745} C_VEL
LIN {X 0,Y 587.213,Z 781.895,A -85,B 0,C 180,E1 -1533.775,E2 -1533.775} C_VEL
LIN {X 0,Y 587.147,Z 777.948,A -85,B 0,C 180,E1 -1534.807,E2 -1534.807} C_VEL
LIN {X 0,Y 587.217,Z 771.876,A -85,B 0,C 180,E1 -1536.011,E2 -1536.011} C_VEL
LIN {X 0,Y 587.245,Z 765.234,A -85,B 0,C 180,E1 -1537.046,E2 -1537.046} C_VEL
LIN {X 0,Y 587.3,Z 756.988,A -85,B 0,C 180,E1 -1538.083,E2 -1538.083} C_VEL
LIN {X 0,Y 587.343,Z 748.535,A -85,B 0,C 180,E1 -1538.949,E2 -1538.949} C_VEL
LIN {X 0,Y 587.421,Z 738.091,A -85,B 0,C 180,E1 -1539.816,E2 -1539.816} C_VEL
LIN {X 0,Y 587.493,Z 727.755,A -85,B 0,C 180,E1 -1540.512,E2 -1540.512} C_VEL
LIN {X 0,Y 587.533,Z 716.125,A -85,B 0,C 180,E1 -1541.135,E2 -1541.135} C_VEL
LIN {X 0,Y 587.591,Z 703.669,A -85,B 0,C 180,E1 -1541.638,E2 -1541.638} C_VEL
LIN {X 0,Y 587.694,Z 690.427,A -85,B 0,C 180,E1 -1542.014,E2 -1542.014} C_VEL
LIN {X 0,Y 587.546,Z 683.637,A -85,B 0,C 180,E1 -1542.154,E2 -1542.154} C_VEL
LIN {X 0,Y 587.197,Z 681.491,A -85,B 0,C 180,E1 -1542.2,E2 -1542.2} C_VEL
LIN {X 0,Y 587.222,Z 672.934,A -85,B 0,C 180,E1 -1544.911,E2 -1544.911} C_VEL
LIN {X 0,Y 587.278,Z 664.03,A -85,B 0,C 180,E1 -1547.768,E2 -1547.768} C_VEL
LIN {X 0,Y 587.3,Z 655.141,A -85,B 0,C 180,E1 -1550.667,E2 -1550.667} C_VEL
LIN {X 0,Y 587.331,Z 646.221,A -85,B 0,C 180,E1 -1553.632,E2 -1553.632} C_VEL
LIN {X 0,Y 587.366,Z 638.43,A -85,B 0,C 180,E1 -1556.277,E2 -1556.277} C_VEL
LIN {X 0,Y 587.41,Z 630.185,A -85,B 0,C 180,E1 -1559.143,E2 -1559.143} C_VEL
LIN {X 0,Y 587.403,Z 623.94,A -85,B 0,C 180,E1 -1561.363,E2 -1561.363} C_VEL
LIN {X 0,Y 587.444,Z 617.158,A -85,B 0,C 180,E1 -1563.801,E2 -1563.801} C_VEL
LIN {X 0,Y 587.507,Z 612.508,A -85,B 0,C 180,E1 -1565.566,E2 -1565.566} C_VEL
LIN {X 0,Y 587.316,Z 611.331,A -85,B 0,C 180,E1 -1566.11,E2 -1566.11} C_VEL
LIN {X 0,Y 587.333,Z 611.327,A -85,B 0,C 180,E1 -1568.479,E2 -1568.479} C_VEL
LIN {X 0,Y 587.339,Z 611.328,A -85,B 0,C 180,E1 -1571.157,E2 -1571.157} C_VEL
LIN {X 0,Y 587.337,Z 611.327,A -85,B 0,C 180,E1 -1574.114,E2 -1574.114} C_VEL
LIN {X 0,Y 587.315,Z 611.329,A -85,B 0,C 180,E1 -1576.993,E2 -1576.993} C_VEL
LIN {X 0,Y 587.319,Z 611.328,A -85,B 0,C 180,E1 -1579.746,E2 -1579.746} C_VEL
LIN {X 0,Y 587.345,Z 611.327,A -85,B 0,C 180,E1 -1582.392,E2 -1582.392} C_VEL
LIN {X 0,Y 587.356,Z 611.324,A -85,B 0,C 180,E1 -1585.651,E2 -1585.651} C_VEL
LIN {X 0,Y 587.354,Z 611.325,A -85,B 0,C 180,E1 -1588.232,E2 -1588.232} C_VEL
LIN {X 0,Y 587.351,Z 611.324,A -85,B 0,C 180,E1 -1590.866,E2 -1590.866} C_VEL
LIN {X 0,Y 587.361,Z 611.323,A -85,B 0,C 180,E1 -1593.819,E2 -1593.819} C_VEL
LIN {X 0,Y 587.337,Z 611.325,A -85,B 0,C 180,E1 -1595.993,E2 -1595.993} C_VEL
LIN {X 0,Y 587.326,Z 611.328,A -85,B 0,C 180,E1 -1598.226,E2 -1598.226} C_VEL
LIN {X 0,Y 587.353,Z 611.324,A -85,B 0,C 180,E1 -1601.151,E2 -1601.151} C_VEL
LIN {X 0,Y 587.328,Z 611.327,A -85,B 0,C 180,E1 -1604.025,E2 -1604.025} C_VEL
LIN {X 0,Y 587.361,Z 611.323,A -85,B 0,C 180,E1 -1606.154,E2 -1606.154} C_VEL
LIN {X 0,Y 587.344,Z 611.325,A -85,B 0,C 180,E1 -1608.962,E2 -1608.962} C_VEL
LIN {X 0,Y 587.37,Z 611.323,A -85,B 0,C 180,E1 -1611.745,E2 -1611.745} C_VEL
LIN {X 0,Y 587.362,Z 611.323,A -85,B 0,C 180,E1 -1614.507,E2 -1614.507} C_VEL
LIN {X 0,Y 587.376,Z 611.321,A -85,B 0,C 180,E1 -1617.257,E2 -1617.257} C_VEL
LIN {X 0,Y 587.382,Z 611.321,A -85,B 0,C 180,E1 -1620,E2 -1620} C_VEL
LIN {X 0,Y 587.382,Z 611.323,A -85,B 0,C 180,E1 -1622.743,E2 -1622.743} C_VEL
LIN {X 0,Y 587.362,Z 611.323,A -85,B 0,C 180,E1 -1625.493,E2 -1625.493} C_VEL
LIN {X 0,Y 587.372,Z 611.322,A -85,B 0,C 180,E1 -1628.255,E2 -1628.255} C_VEL
LIN {X 0,Y 587.289,Z 611.333,A -85,B 0,C 180,E1 -1629.645,E2 -1629.645} C_VEL
LIN {X 0,Y 587.35,Z 613.615,A -85,B 0,C 180,E1 -1631.134,E2 -1631.134} C_VEL
LIN {X 0,Y 587.265,Z 618.699,A -85,B 0,C 180,E1 -1634.221,E2 -1634.221} C_VEL
LIN {X 0,Y 587.256,Z 623.193,A -85,B 0,C 180,E1 -1636.784,E2 -1636.784} C_VEL
LIN {X 0,Y 587.226,Z 625.666,A -85,B 0,C 180,E1 -1638.166,E2 -1638.166} C_VEL
LIN {X 0,Y 586.549,Z 626.74,A -85,B 0,C 180,E1 -1638.729,E2 -1638.729} C_VEL
LIN {X 0,Y 583.66,Z 628.633,A -85,B 0,C 180,E1 -1639.639,E2 -1639.639} C_VEL
LIN {X 0,Y 581.242,Z 630.16,A -85,B 0,C 180,E1 -1640.37,E2 -1640.37} C_VEL
LIN {X 0,Y 580.236,Z 631.271,A -85,B 0,C 180,E1 -1640.937,E2 -1640.937} C_VEL
LIN {X 0,Y 580.172,Z 631.625,A -85,B 0,C 180,E1 -1641.129,E2 -1641.129} C_VEL
LIN {X 0,Y 580.127,Z 636.105,A -85,B 0,C 180,E1 -1643.565,E2 -1643.565} C_VEL
LIN {X 0,Y 580.087,Z 641.853,A -85,B 0,C 180,E1 -1646.633,E2 -1646.633} C_VEL
LIN {X 0,Y 580.084,Z 646.876,A -85,B 0,C 180,E1 -1649.271,E2 -1649.271} C_VEL
LIN {X 0,Y 580.049,Z 652.561,A -85,B 0,C 180,E1 -1652.216,E2 -1652.216} C_VEL
LIN {X 0,Y 580.068,Z 653.558,A -85,B 0,C 180,E1 -1652.729,E2 -1652.729} C_VEL
LIN {X 0,Y 580.773,Z 659.594,A -85,B 0,C 180,E1 -1652.865,E2 -1652.865} C_VEL
LIN {X 0,Y 580.688,Z 672.516,A -85,B 0,C 180,E1 -1653.228,E2 -1653.228} C_VEL
LIN {X 0,Y 580.566,Z 684.566,A -85,B 0,C 180,E1 -1653.704,E2 -1653.704} C_VEL
LIN {X 0,Y 580.515,Z 695.33,A -85,B 0,C 180,E1 -1654.26,E2 -1654.26} C_VEL
LIN {X 0,Y 580.435,Z 706.691,A -85,B 0,C 180,E1 -1655.004,E2 -1655.004} C_VEL
LIN {X 0,Y 580.344,Z 717.396,A -85,B 0,C 180,E1 -1655.884,E2 -1655.884} C_VEL
LIN {X 0,Y 580.243,Z 726.391,A -85,B 0,C 180,E1 -1656.794,E2 -1656.794} C_VEL
LIN {X 0,Y 580.168,Z 734.891,A -85,B 0,C 180,E1 -1657.864,E2 -1657.864} C_VEL
LIN {X 0,Y 580.142,Z 741.084,A -85,B 0,C 180,E1 -1658.823,E2 -1658.823} C_VEL
LIN {X 0,Y 580.113,Z 746.903,A -85,B 0,C 180,E1 -1659.948,E2 -1659.948} C_VEL
LIN {X 0,Y 580.071,Z 750.631,A -85,B 0,C 180,E1 -1660.863,E2 -1660.863} C_VEL
LIN {X 0,Y 580.091,Z 753.583,A -85,B 0,C 180,E1 -1661.786,E2 -1661.786} C_VEL
LIN {X 0,Y 580.058,Z 755.772,A -85,B 0,C 180,E1 -1662.727,E2 -1662.727} C_VEL
LIN {X 0,Y 580.028,Z 757.214,A -85,B 0,C 180,E1 -1663.682,E2 -1663.682} C_VEL
LIN {X 0,Y 580.037,Z 757.917,A -85,B 0,C 180,E1 -1664.649,E2 -1664.649} C_VEL
LIN {X 0,Y 580.041,Z 757.855,A -85,B 0,C 180,E1 -1665.633,E2 -1665.633} C_VEL
LIN {X 0,Y 580.033,Z 756.955,A -85,B 0,C 180,E1 -1666.635,E2 -1666.635} C_VEL
LIN {X 0,Y 580.066,Z 755.175,A -85,B 0,C 180,E1 -1667.652,E2 -1667.652} C_VEL
LIN {X 0,Y 580.074,Z 752.426,A -85,B 0,C 180,E1 -1668.692,E2 -1668.692} C_VEL
LIN {X 0,Y 580.12,Z 748.603,A -85,B 0,C 180,E1 -1669.75,E2 -1669.75} C_VEL
LIN {X 0,Y 580.133,Z 742.877,A -85,B 0,C 180,E1 -1670.953,E2 -1670.953} C_VEL
LIN {X 0,Y 580.168,Z 735.526,A -85,B 0,C 180,E1 -1672.137,E2 -1672.137} C_VEL
LIN {X 0,Y 580.242,Z 727.163,A -85,B 0,C 180,E1 -1673.207,E2 -1673.207} C_VEL
LIN {X 0,Y 580.339,Z 718.375,A -85,B 0,C 180,E1 -1674.118,E2 -1674.118} C_VEL
LIN {X 0,Y 580.436,Z 707.884,A -85,B 0,C 180,E1 -1674.997,E2 -1674.997} C_VEL
LIN {X 0,Y 580.5,Z 696.881,A -85,B 0,C 180,E1 -1675.739,E2 -1675.739} C_VEL
LIN {X 0,Y 580.604,Z 684.974,A -85,B 0,C 180,E1 -1676.367,E2 -1676.367} C_VEL
LIN {X 0,Y 580.688,Z 671.974,A -85,B 0,C 180,E1 -1676.881,E2 -1676.881} C_VEL
LIN {X 0,Y 580.761,Z 659.074,A -85,B 0,C 180,E1 -1677.237,E2 -1677.237} C_VEL
LIN {X 0,Y 580.063,Z 653.533,A -85,B 0,C 180,E1 -1677.374,E2 -1677.374} C_VEL
LIN {X 0,Y 580.061,Z 648.037,A -85,B 0,C 180,E1 -1680.214,E2 -1680.214} C_VEL
LIN {X 0,Y 580.074,Z 643.502,A -85,B 0,C 180,E1 -1682.587,E2 -1682.587} C_VEL
LIN {X 0,Y 580.1,Z 638.354,A -85,B 0,C 180,E1 -1685.318,E2 -1685.318} C_VEL
LIN {X 0,Y 580.127,Z 633.493,A -85,B 0,C 180,E1 -1687.941,E2 -1687.941} C_VEL
LIN {X 0,Y 580.184,Z 628.104,A -85,B 0,C 180,E1 -1690.909,E2 -1690.909} C_VEL
LIN {X 0,Y 580.185,Z 622.947,A -85,B 0,C 180,E1 -1693.823,E2 -1693.823} C_VEL
LIN {X 0,Y 580.206,Z 618.142,A -85,B 0,C 180,E1 -1696.694,E2 -1696.694} C_VEL
LIN {X 0,Y 580.282,Z 613.352,A -85,B 0,C 180,E1 -1699.533,E2 -1699.533} C_VEL
LIN {X 0,Y 580.205,Z 612.216,A -85,B 0,C 180,E1 -1700.236,E2 -1700.236} C_VEL
LIN {X 0,Y 580.334,Z 612.198,A -85,B 0,C 180,E1 -1702.344,E2 -1702.344} C_VEL
LIN {X 0,Y 580.331,Z 612.199,A -85,B 0,C 180,E1 -1705.137,E2 -1705.137} C_VEL
LIN {X 0,Y 580.346,Z 612.195,A -85,B 0,C 180,E1 -1707.918,E2 -1707.918} C_VEL
LIN {X 0,Y 580.368,Z 612.195,A -85,B 0,C 180,E1 -1710.694,E2 -1710.694} C_VEL
LIN {X 0,Y 580.289,Z 612.203,A -85,B 0,C 180,E1 -1713.471,E2 -1713.471} C_VEL
LIN {X 0,Y 580.326,Z 612.201,A -85,B 0,C 180,E1 -1715.559,E2 -1715.559} C_VEL
LIN {X 0,Y 580.324,Z 612.199,A -85,B 0,C 180,E1 -1718.356,E2 -1718.356} C_VEL
LIN {X 0,Y 580.177,Z 612.442,A -85,B 0,C 180,E1 -1719.588,E2 -1719.588} C_VEL
LIN {X 0,Y 580.184,Z 616.775,A -85,B 0,C 180,E1 -1721.883,E2 -1721.883} C_VEL
LIN {X 0,Y 580.179,Z 622.019,A -85,B 0,C 180,E1 -1724.737,E2 -1724.737} C_VEL
LIN {X 0,Y 580.152,Z 627.119,A -85,B 0,C 180,E1 -1727.629,E2 -1727.629} C_VEL
LIN {X 0,Y 580.12,Z 631.083,A -85,B 0,C 180,E1 -1729.828,E2 -1729.828} C_VEL
LIN {X 0,Y 580.137,Z 636.557,A -85,B 0,C 180,E1 -1732.809,E2 -1732.809} C_VEL
LIN {X 0,Y 580.082,Z 640.828,A -85,B 0,C 180,E1 -1735.09,E2 -1735.09} C_VEL
LIN {X 0,Y 580.072,Z 646.004,A -85,B 0,C 180,E1 -1737.816,E2 -1737.816} C_VEL
LIN {X 0,Y 580.059,Z 651.475,A -85,B 0,C 180,E1 -1740.656,E2 -1740.656} C_VEL
LIN {X 0,Y 580.058,Z 653.541,A -85,B 0,C 180,E1 -1741.721,E2 -1741.721} C_VEL
LIN {X 0,Y 580.773,Z 659.563,A -85,B 0,C 180,E1 -1741.864,E2 -1741.864} C_VEL
LIN {X 0,Y 580.694,Z 672.462,A -85,B 0,C 180,E1 -1742.227,E2 -1742.227} C_VEL
LIN {X 0,Y 580.626,Z 684.25,A -85,B 0,C 180,E1 -1742.693,E2 -1742.693} C_VEL
LIN {X 0,Y 580.471,Z 695.449,A -85,B 0,C 180,E1 -1743.269,E2 -1743.269} C_VEL
LIN {X 0,Y 580.415,Z 706.007,A -85,B 0,C 180,E1 -1743.952,E2 -1743.952} C_VEL
LIN {X 0,Y 580.32,Z 716.472,A -85,B 0,C 180,E1 -1744.799,E2 -1744.799} C_VEL
LIN {X 0,Y 580.258,Z 726.031,A -85,B 0,C 180,E1 -1745.757,E2 -1745.757} C_VEL
LIN {X 0,Y 580.163,Z 733.421,A -85,B 0,C 180,E1 -1746.662,E2 -1746.662} C_VEL
LIN {X 0,Y 580.11,Z 740.156,A -85,B 0,C 180,E1 -1747.665,E2 -1747.665} C_VEL
LIN {X 0,Y 580.114,Z 746.339,A -85,B 0,C 180,E1 -1748.824,E2 -1748.824} C_VEL
LIN {X 0,Y 580.088,Z 750.943,A -85,B 0,C 180,E1 -1749.949,E2 -1749.949} C_VEL
LIN {X 0,Y 580.039,Z 754.87,A -85,B 0,C 180,E1 -1751.304,E2 -1751.304} C_VEL
LIN {X 0,Y 580.063,Z 756.795,A -85,B 0,C 180,E1 -1752.347,E2 -1752.347} C_VEL
LIN {X 0,Y 580.025,Z 757.925,A -85,B 0,C 180,E1 -1753.681,E2 -1753.681} C_VEL
LIN {X 0,Y 580.039,Z 757.827,A -85,B 0,C 180,E1 -1754.648,E2 -1754.648} C_VEL
LIN {X 0,Y 580.039,Z 756.94,A -85,B 0,C 180,E1 -1755.632,E2 -1755.632} C_VEL
LIN {X 0,Y 580.032,Z 755.202,A -85,B 0,C 180,E1 -1756.634,E2 -1756.634} C_VEL
LIN {X 0,Y 580.084,Z 752.543,A -85,B 0,C 180,E1 -1757.649,E2 -1757.649} C_VEL
LIN {X 0,Y 580.078,Z 748.827,A -85,B 0,C 180,E1 -1758.691,E2 -1758.691} C_VEL
LIN {X 0,Y 580.127,Z 743.936,A -85,B 0,C 180,E1 -1759.748,E2 -1759.748} C_VEL
LIN {X 0,Y 580.183,Z 736.782,A -85,B 0,C 180,E1 -1760.957,E2 -1760.957} C_VEL
LIN {X 0,Y 580.248,Z 727.941,A -85,B 0,C 180,E1 -1762.115,E2 -1762.115} C_VEL
LIN {X 0,Y 580.306,Z 718.914,A -85,B 0,C 180,E1 -1763.064,E2 -1763.064} C_VEL
LIN {X 0,Y 580.397,Z 708.579,A -85,B 0,C 180,E1 -1763.945,E2 -1763.945} C_VEL
LIN {X 0,Y 580.479,Z 697.828,A -85,B 0,C 180,E1 -1764.681,E2 -1764.681} C_VEL
LIN {X 0,Y 580.598,Z 685.851,A -85,B 0,C 180,E1 -1765.325,E2 -1765.325} C_VEL
LIN {X 0,Y 580.676,Z 674.21,A -85,B 0,C 180,E1 -1765.803,E2 -1765.803} C_VEL
LIN {X 0,Y 580.767,Z 661.665,A -85,B 0,C 180,E1 -1766.175,E2 -1766.175} C_VEL
LIN {X 0,Y 580.496,Z 656.332,A -85,B 0,C 180,E1 -1766.297,E2 -1766.297} C_VEL
LIN {X 0,Y 580.068,Z 653.541,A -85,B 0,C 180,E1 -1766.369,E2 -1766.369} C_VEL
LIN {X 0,Y 580.069,Z 647.658,A -85,B 0,C 180,E1 -1769.412,E2 -1769.412} C_VEL
LIN {X 0,Y 580.07,Z 642.372,A -85,B 0,C 180,E1 -1772.183,E2 -1772.183} C_VEL
LIN {X 0,Y 580.102,Z 638.684,A -85,B 0,C 180,E1 -1774.142,E2 -1774.142} C_VEL
LIN {X 0,Y 580.134,Z 633.336,A -85,B 0,C 180,E1 -1777.027,E2 -1777.027} C_VEL
LIN {X 0,Y 580.159,Z 628.962,A -85,B 0,C 180,E1 -1779.433,E2 -1779.433} C_VEL
LIN {X 0,Y 580.165,Z 625.023,A -85,B 0,C 180,E1 -1781.642,E2 -1781.642} C_VEL
LIN {X 0,Y 580.176,Z 621.117,A -85,B 0,C 180,E1 -1783.823,E2 -1783.823} C_VEL
LIN {X 0,Y 580.177,Z 615.62,A -85,B 0,C 180,E1 -1786.694,E2 -1786.694} C_VEL
LIN {X 0,Y 580.173,Z 612.22,A -85,B 0,C 180,E1 -1788.47,E2 -1788.47} C_VEL
LIN {X 0,Y 580.293,Z 612.205,A -85,B 0,C 180,E1 -1790.941,E2 -1790.941} C_VEL
LIN {X 0,Y 580.348,Z 612.198,A -85,B 0,C 180,E1 -1793.22,E2 -1793.22} C_VEL
LIN {X 0,Y 580.275,Z 612.206,A -85,B 0,C 180,E1 -1795.833,E2 -1795.833} C_VEL
LIN {X 0,Y 580.336,Z 612.198,A -85,B 0,C 180,E1 -1797.918,E2 -1797.918} C_VEL
LIN {X 0,Y 580.363,Z 612.195,A -85,B 0,C 180,E1 -1800.694,E2 -1800.694} C_VEL
LIN {X 0,Y 580.289,Z 612.206,A -85,B 0,C 180,E1 -1803.472,E2 -1803.472} C_VEL
LIN {X 0,Y 580.325,Z 612.201,A -85,B 0,C 180,E1 -1805.56,E2 -1805.56} C_VEL
LIN {X 0,Y 580.332,Z 612.199,A -85,B 0,C 180,E1 -1808.356,E2 -1808.356} C_VEL
LIN {X 0,Y 580.33,Z 612.198,A -85,B 0,C 180,E1 -1811.208,E2 -1811.208} C_VEL
LIN {X 0,Y 580.312,Z 612.201,A -85,B 0,C 180,E1 -1814.339,E2 -1814.339} C_VEL
LIN {X 0,Y 580.308,Z 612.203,A -85,B 0,C 180,E1 -1816.914,E2 -1816.914} C_VEL
LIN {X 0,Y 580.303,Z 612.204,A -85,B 0,C 180,E1 -1819.822,E2 -1819.822} C_VEL
LIN {X 0,Y 580.293,Z 612.205,A -85,B 0,C 180,E1 -1822.803,E2 -1822.803} C_VEL
LIN {X 0,Y 580.307,Z 612.203,A -85,B 0,C 180,E1 -1825.08,E2 -1825.08} C_VEL
LIN {X 0,Y 580.317,Z 612.201,A -85,B 0,C 180,E1 -1827.863,E2 -1827.863} C_VEL
LIN {X 0,Y 580.297,Z 612.202,A -85,B 0,C 180,E1 -1830.698,E2 -1830.698} C_VEL
LIN {X 0,Y 580.303,Z 612.204,A -85,B 0,C 180,E1 -1833.317,E2 -1833.317} C_VEL
LIN {X 0,Y 580.274,Z 612.205,A -85,B 0,C 180,E1 -1835.761,E2 -1835.761} C_VEL
LIN {X 0,Y 580.286,Z 612.204,A -85,B 0,C 180,E1 -1838.147,E2 -1838.147} C_VEL
LIN {X 0,Y 580.298,Z 612.203,A -85,B 0,C 180,E1 -1840.844,E2 -1840.844} C_VEL
LIN {X 0,Y 580.271,Z 612.207,A -85,B 0,C 180,E1 -1843.659,E2 -1843.659} C_VEL
LIN {X 0,Y 580.276,Z 612.208,A -85,B 0,C 180,E1 -1846.61,E2 -1846.61} C_VEL
LIN {X 0,Y 580.298,Z 612.203,A -85,B 0,C 180,E1 -1849.157,E2 -1849.157} C_VEL
LIN {X 0,Y 580.29,Z 612.205,A -85,B 0,C 180,E1 -1851.927,E2 -1851.927} C_VEL
LIN {X 0,Y 580.338,Z 612.349,A -85,B 0,C 180,E1 -1853.855,E2 -1853.855} C_VEL
LIN {X 0,Y 580.56,Z 616.321,A -85,B 0,C 180,E1 -1855.405,E2 -1855.405} C_VEL
LIN {X 0,Y 580.472,Z 623.162,A -85,B 0,C 180,E1 -1857.943,E2 -1857.943} C_VEL
LIN {X 0,Y 580.382,Z 630.765,A -85,B 0,C 180,E1 -1860.677,E2 -1860.677} C_VEL
LIN {X 0,Y 580.348,Z 639.221,A -85,B 0,C 180,E1 -1863.655,E2 -1863.655} C_VEL
LIN {X 0,Y 580.288,Z 647.336,A -85,B 0,C 180,E1 -1866.443,E2 -1866.443} C_VEL
LIN {X 0,Y 580.242,Z 656.241,A -85,B 0,C 180,E1 -1869.436,E2 -1869.436} C_VEL
LIN {X 0,Y 580.202,Z 665.145,A -85,B 0,C 180,E1 -1872.373,E2 -1872.373} C_VEL
LIN {X 0,Y 580.154,Z 674.049,A -85,B 0,C 180,E1 -1875.263,E2 -1875.263} C_VEL
LIN {X 0,Y 580.127,Z 681.493,A -85,B 0,C 180,E1 -1877.649,E2 -1877.649} C_VEL
LIN {X 0,Y 580.823,Z 687.39,A -85,B 0,C 180,E1 -1877.775,E2 -1877.775} C_VEL
LIN {X 0,Y 580.718,Z 699.51,A -85,B 0,C 180,E1 -1878.083,E2 -1878.083} C_VEL
LIN {X 0,Y 580.624,Z 711.328,A -85,B 0,C 180,E1 -1878.515,E2 -1878.515} C_VEL
LIN {X 0,Y 580.52,Z 723.217,A -85,B 0,C 180,E1 -1879.096,E2 -1879.096} C_VEL
LIN {X 0,Y 580.45,Z 734.484,A -85,B 0,C 180,E1 -1879.801,E2 -1879.801} C_VEL
LIN {X 0,Y 580.352,Z 744.651,A -85,B 0,C 180,E1 -1880.591,E2 -1880.591} C_VEL
LIN {X 0,Y 580.279,Z 753.79,A -85,B 0,C 180,E1 -1881.468,E2 -1881.468} C_VEL
LIN {X 0,Y 580.199,Z 762.693,A -85,B 0,C 180,E1 -1882.518,E2 -1882.518} C_VEL
LIN {X 0,Y 580.12,Z 769.464,A -85,B 0,C 180,E1 -1883.505,E2 -1883.505} C_VEL
LIN {X 0,Y 580.139,Z 774.682,A -85,B 0,C 180,E1 -1884.439,E2 -1884.439} C_VEL
LIN {X 0,Y 580.108,Z 779.373,A -85,B 0,C 180,E1 -1885.484,E2 -1885.484} C_VEL
LIN {X 0,Y 580.123,Z 782.958,A -85,B 0,C 180,E1 -1886.528,E2 -1886.528} C_VEL
LIN {X 0,Y 580.043,Z 784.809,A -85,B 0,C 180,E1 -1887.222,E2 -1887.222} C_VEL
LIN {X 0,Y 580.039,Z 786.201,A -85,B 0,C 180,E1 -1887.917,E2 -1887.917} C_VEL
LIN {X 0,Y 580.04,Z 787.784,A -85,B 0,C 180,E1 -1889.306,E2 -1889.306} C_VEL
LIN {X 0,Y 580.037,Z 788,A -85,B 0,C 180,E1 -1890,E2 -1890} C_VEL
LIN {X 0,Y 580.046,Z 787.185,A -85,B 0,C 180,E1 -1891.389,E2 -1891.389} C_VEL
LIN {X 0,Y 580.039,Z 786.201,A -85,B 0,C 180,E1 -1892.083,E2 -1892.083} C_VEL
LIN {X 0,Y 580.043,Z 784.809,A -85,B 0,C 180,E1 -1892.778,E2 -1892.778} C_VEL
LIN {X 0,Y 580.11,Z 781.895,A -85,B 0,C 180,E1 -1893.821,E2 -1893.821} C_VEL
LIN {X 0,Y 580.053,Z 777.948,A -85,B 0,C 180,E1 -1894.866,E2 -1894.866} C_VEL
LIN {X 0,Y 580.139,Z 771.876,A -85,B 0,C 180,E1 -1896.085,E2 -1896.085} C_VEL
LIN {X 0,Y 580.184,Z 765.235,A -85,B 0,C 180,E1 -1897.133,E2 -1897.133} C_VEL
LIN {X 0,Y 580.251,Z 756.988,A -85,B 0,C 180,E1 -1898.182,E2 -1898.182} C_VEL
LIN {X 0,Y 580.308,Z 748.535,A -85,B 0,C 180,E1 -1899.059,E2 -1899.059} C_VEL
LIN {X 0,Y 580.417,Z 738.092,A -85,B 0,C 180,E1 -1899.936,E2 -1899.936} C_VEL
LIN {X 0,Y 580.498,Z 727.754,A -85,B 0,C 180,E1 -1900.64,E2 -1900.64} C_VEL
LIN {X 0,Y 580.564,Z 716.587,A -85,B 0,C 180,E1 -1901.248,E2 -1901.248} C_VEL
LIN {X 0,Y 580.624,Z 704.76,A -85,B 0,C 180,E1 -1901.742,E2 -1901.742} C_VEL
LIN {X 0,Y 580.76,Z 691.341,A -85,B 0,C 180,E1 -1902.138,E2 -1902.138} C_VEL
LIN {X 0,Y 580.563,Z 684.363,A -85,B 0,C 180,E1 -1902.289,E2 -1902.289} C_VEL
LIN {X 0,Y 580.128,Z 681.491,A -85,B 0,C 180,E1 -1902.351,E2 -1902.351} C_VEL
LIN {X 0,Y 580.156,Z 672.934,A -85,B 0,C 180,E1 -1905.097,E2 -1905.097} C_VEL
LIN {X 0,Y 580.207,Z 664.03,A -85,B 0,C 180,E1 -1907.992,E2 -1907.992} C_VEL
LIN {X 0,Y 580.243,Z 656.239,A -85,B 0,C 180,E1 -1910.564,E2 -1910.564} C_VEL
LIN {X 0,Y 580.289,Z 647.334,A -85,B 0,C 180,E1 -1913.558,E2 -1913.558} C_VEL
LIN {X 0,Y 580.35,Z 639.219,A -85,B 0,C 180,E1 -1916.345,E2 -1916.345} C_VEL
LIN {X 0,Y 580.384,Z 630.764,A -85,B 0,C 180,E1 -1919.324,E2 -1919.324} C_VEL
LIN {X 0,Y 580.398,Z 625.007,A -85,B 0,C 180,E1 -1921.378,E2 -1921.378} C_VEL
LIN {X 0,Y 580.46,Z 618.235,A -85,B 0,C 180,E1 -1923.845,E2 -1923.845} C_VEL
LIN {X 0,Y 580.462,Z 613.222,A -85,B 0,C 180,E1 -1925.785,E2 -1925.785} C_VEL
LIN {X 0,Y 580.273,Z 612.208,A -85,B 0,C 180,E1 -1926.233,E2 -1926.233} C_VEL
LIN {X 0,Y 580.3,Z 612.205,A -85,B 0,C 180,E1 -1929.185,E2 -1929.185} C_VEL
LIN {X 0,Y 580.317,Z 612.201,A -85,B 0,C 180,E1 -1931.766,E2 -1931.766} C_VEL
LIN {X 0,Y 580.265,Z 612.207,A -85,B 0,C 180,E1 -1934.626,E2 -1934.626} C_VEL
LIN {X 0,Y 580.288,Z 612.204,A -85,B 0,C 180,E1 -1937.628,E2 -1937.628} C_VEL
LIN {X 0,Y 580.296,Z 612.204,A -85,B 0,C 180,E1 -1940.067,E2 -1940.067} C_VEL
LIN {X 0,Y 580.3,Z 612.203,A -85,B 0,C 180,E1 -1943.066,E2 -1943.066} C_VEL
LIN {X 0,Y 580.321,Z 612.2,A -85,B 0,C 180,E1 -1946.145,E2 -1946.145} C_VEL
LIN {X 0,Y 580.29,Z 612.205,A -85,B 0,C 180,E1 -1948.615,E2 -1948.615} C_VEL
LIN {X 0,Y 580.294,Z 612.203,A -85,B 0,C 180,E1 -1951.024,E2 -1951.024} C_VEL
LIN {X 0,Y 580.293,Z 612.204,A -85,B 0,C 180,E1 -1953.666,E2 -1953.666} C_VEL
LIN {X 0,Y 580.302,Z 612.203,A -85,B 0,C 180,E1 -1955.684,E2 -1955.684} C_VEL
LIN {X 0,Y 580.276,Z 612.205,A -85,B 0,C 180,E1 -1957.947,E2 -1957.947} C_VEL
LIN {X 0,Y 580.321,Z 612.2,A -85,B 0,C 180,E1 -1960.914,E2 -1960.914} C_VEL
LIN {X 0,Y 580.282,Z 612.205,A -85,B 0,C 180,E1 -1963.826,E2 -1963.826} C_VEL
LIN {X 0,Y 580.327,Z 612.199,A -85,B 0,C 180,E1 -1965.983,E2 -1965.983} C_VEL
LIN {X 0,Y 580.306,Z 612.203,A -85,B 0,C 180,E1 -1968.827,E2 -1968.827} C_VEL
LIN {X 0,Y 580.335,Z 612.2,A -85,B 0,C 180,E1 -1971.644,E2 -1971.644} C_VEL
LIN {X 0,Y 580.328,Z 612.199,A -85,B 0,C 180,E1 -1974.44,E2 -1974.44} C_VEL
LIN {X 0,Y 580.343,Z 612.197,A -85,B 0,C 180,E1 -1977.224,E2 -1977.224} C_VEL
LIN {X 0,Y 580.352,Z 612.197,A -85,B 0,C 180,E1 -1980,E2 -1980} C_VEL
LIN {X 0,Y 580.347,Z 612.199,A -85,B 0,C 180,E1 -1982.777,E2 -1982.777} C_VEL
LIN {X 0,Y 580.328,Z 612.2,A -85,B 0,C 180,E1 -1985.56,E2 -1985.56} C_VEL
LIN {X 0,Y 580.336,Z 612.198,A -85,B 0,C 180,E1 -1988.356,E2 -1988.356} C_VEL
LIN {X 0,Y 580.226,Z 612.214,A -85,B 0,C 180,E1 -1989.763,E2 -1989.763} C_VEL
LIN {X 0,Y 580.237,Z 615.701,A -85,B 0,C 180,E1 -1991.883,E2 -1991.883} C_VEL
LIN {X 0,Y 580.17,Z 620.304,A -85,B 0,C 180,E1 -1994.737,E2 -1994.737} C_VEL
LIN {X 0,Y 580.161,Z 625.342,A -85,B 0,C 180,E1 -1997.629,E2 -1997.629} C_VEL
LIN {X 0,Y 580.136,Z 629.272,A -85,B 0,C 180,E1 -1999.828,E2 -1999.828} C_VEL
LIN {X 0,Y 580.172,Z 631.625,A -85,B 0,C 180,E1 -2001.129,E2 -2001.129} C_VEL
LIN {X 0,Y 579.543,Z 632.714,A -85,B 0,C 180,E1 -2001.698,E2 -2001.698} C_VEL
LIN {X 0,Y 576.66,Z 634.619,A -85,B 0,C 180,E1 -2002.62,E2 -2002.62} C_VEL
LIN {X 0,Y 574.188,Z 636.159,A -85,B 0,C 180,E1 -2003.361,E2 -2003.361} C_VEL
LIN {X 0,Y 573.113,Z 637.288,A -85,B 0,C 180,E1 -2003.934,E2 -2003.934} C_VEL
LIN {X 0,Y 573.02,Z 637.652,A -85,B 0,C 180,E1 -2004.129,E2 -2004.129} C_VEL
LIN {X 0,Y 573.008,Z 642.957,A -85,B 0,C 180,E1 -2006.988,E2 -2006.988} C_VEL
LIN {X 0,Y 572.985,Z 647.578,A -85,B 0,C 180,E1 -2009.442,E2 -2009.442} C_VEL
LIN {X 0,Y 572.986,Z 653.212,A -85,B 0,C 180,E1 -2012.395,E2 -2012.395} C_VEL
LIN {X 0,Y 572.989,Z 653.718,A -85,B 0,C 180,E1 -2012.578,E2 -2012.578} C_VEL
LIN {X 0,Y 573.849,Z 660.473,A -85,B 0,C 180,E1 -2012.737,E2 -2012.737} C_VEL
LIN {X 0,Y 573.735,Z 672.575,A -85,B 0,C 180,E1 -2013.084,E2 -2013.084} C_VEL
LIN {X 0,Y 573.595,Z 684.779,A -85,B 0,C 180,E1 -2013.574,E2 -2013.574} C_VEL
LIN {X 0,Y 573.502,Z 696.775,A -85,B 0,C 180,E1 -2014.213,E2 -2014.213} C_VEL
LIN {X 0,Y 573.427,Z 707.616,A -85,B 0,C 180,E1 -2014.95,E2 -2014.95} C_VEL
LIN {X 0,Y 573.296,Z 717.731,A -85,B 0,C 180,E1 -2015.801,E2 -2015.801} C_VEL
LIN {X 0,Y 573.188,Z 726.537,A -85,B 0,C 180,E1 -2016.708,E2 -2016.708} C_VEL
LIN {X 0,Y 573.105,Z 735.194,A -85,B 0,C 180,E1 -2017.818,E2 -2017.818} C_VEL
LIN {X 0,Y 573.078,Z 740.906,A -85,B 0,C 180,E1 -2018.715,E2 -2018.715} C_VEL
LIN {X 0,Y 573.054,Z 745.706,A -85,B 0,C 180,E1 -2019.623,E2 -2019.623} C_VEL
LIN {X 0,Y 573.008,Z 749.666,A -85,B 0,C 180,E1 -2020.546,E2 -2020.546} C_VEL
LIN {X 0,Y 572.997,Z 754.146,A -85,B 0,C 180,E1 -2021.968,E2 -2021.968} C_VEL
LIN {X 0,Y 572.961,Z 755.596,A -85,B 0,C 180,E1 -2022.611,E2 -2022.611} C_VEL
LIN {X 0,Y 572.928,Z 757.182,A -85,B 0,C 180,E1 -2023.636,E2 -2023.636} C_VEL
LIN {X 0,Y 572.938,Z 757.918,A -85,B 0,C 180,E1 -2024.646,E2 -2024.646} C_VEL
LIN {X 0,Y 572.941,Z 757.857,A -85,B 0,C 180,E1 -2025.638,E2 -2025.638} C_VEL
LIN {X 0,Y 572.935,Z 757.003,A -85,B 0,C 180,E1 -2026.612,E2 -2026.612} C_VEL
LIN {X 0,Y 572.988,Z 755.396,A -85,B 0,C 180,E1 -2027.577,E2 -2027.577} C_VEL
LIN {X 0,Y 573.003,Z 753.071,A -85,B 0,C 180,E1 -2028.523,E2 -2028.523} C_VEL
LIN {X 0,Y 573.012,Z 749.832,A -85,B 0,C 180,E1 -2029.503,E2 -2029.503} C_VEL
LIN {X 0,Y 573.049,Z 745.106,A -85,B 0,C 180,E1 -2030.592,E2 -2030.592} C_VEL
LIN {X 0,Y 573.099,Z 738.921,A -85,B 0,C 180,E1 -2031.706,E2 -2031.706} C_VEL
LIN {X 0,Y 573.149,Z 730.939,A -85,B 0,C 180,E1 -2032.848,E2 -2032.848} C_VEL
LIN {X 0,Y 573.239,Z 722.302,A -85,B 0,C 180,E1 -2033.841,E2 -2033.841} C_VEL
LIN {X 0,Y 573.357,Z 711.649,A -85,B 0,C 180,E1 -2034.823,E2 -2034.823} C_VEL
LIN {X 0,Y 573.477,Z 701.158,A -85,B 0,C 180,E1 -2035.6,E2 -2035.6} C_VEL
LIN {X 0,Y 573.587,Z 689.355,A -85,B 0,C 180,E1 -2036.291,E2 -2036.291} C_VEL
LIN {X 0,Y 573.72,Z 676.566,A -85,B 0,C 180,E1 -2036.862,E2 -2036.862} C_VEL
LIN {X 0,Y 573.834,Z 663.665,A -85,B 0,C 180,E1 -2037.275,E2 -2037.275} C_VEL
LIN {X 0,Y 573.599,Z 657.328,A -85,B 0,C 180,E1 -2037.427,E2 -2037.427} C_VEL
